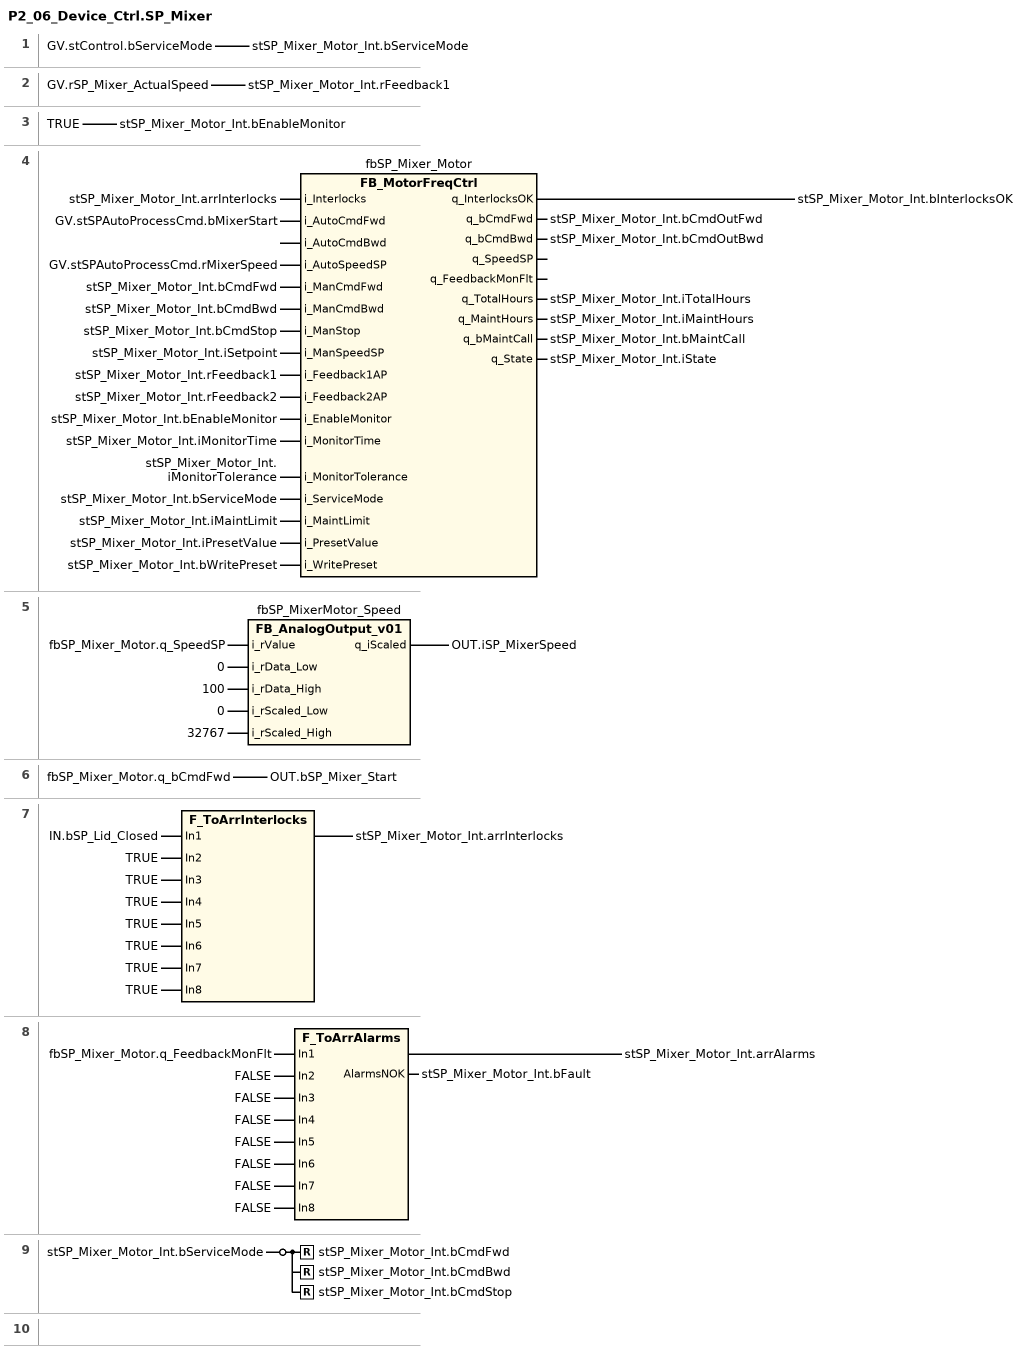
// NETWORK 1
stSP_Mixer_Motor_Int.bServiceMode := GV.stControl.bServiceMode;

// NETWORK 2
stSP_Mixer_Motor_Int.rFeedback1 := GV.rSP_Mixer_ActualSpeed;

// NETWORK 3
stSP_Mixer_Motor_Int.bEnableMonitor := TRUE;

// NETWORK 4
fbSP_Mixer_Motor(
    i_Interlocks := stSP_Mixer_Motor_Int.arrInterlocks,
    i_AutoCmdFwd := GV.stSPAutoProcessCmd.bMixerStart,
    i_AutoSpeedSP := GV.stSPAutoProcessCmd.rMixerSpeed,
    i_ManCmdFwd := stSP_Mixer_Motor_Int.bCmdFwd,
    i_ManCmdBwd := stSP_Mixer_Motor_Int.bCmdBwd,
    i_ManStop := stSP_Mixer_Motor_Int.bCmdStop,
    i_ManSpeedSP := stSP_Mixer_Motor_Int.iSetpoint,
    i_Feedback1AP := stSP_Mixer_Motor_Int.rFeedback1,
    i_Feedback2AP := stSP_Mixer_Motor_Int.rFeedback2,
    i_EnableMonitor := stSP_Mixer_Motor_Int.bEnableMonitor,
    i_MonitorTime := stSP_Mixer_Motor_Int.iMonitorTime,
    i_MonitorTolerance := stSP_Mixer_Motor_Int.iMonitorTolerance,
    i_ServiceMode := stSP_Mixer_Motor_Int.bServiceMode,
    i_MaintLimit := stSP_Mixer_Motor_Int.iMaintLimit,
    i_PresetValue := stSP_Mixer_Motor_Int.iPresetValue,
    i_WritePreset := stSP_Mixer_Motor_Int.bWritePreset,
    q_bCmdFwd => stSP_Mixer_Motor_Int.bCmdOutFwd,
    q_bCmdBwd => stSP_Mixer_Motor_Int.bCmdOutBwd,
    q_TotalHours => stSP_Mixer_Motor_Int.iTotalHours,
    q_MaintHours => stSP_Mixer_Motor_Int.iMaintHours,
    q_bMaintCall => stSP_Mixer_Motor_Int.bMaintCall,
    q_State => stSP_Mixer_Motor_Int.iState); // FB_MotorFreqCtrl
stSP_Mixer_Motor_Int.bInterlocksOK := fbSP_Mixer_Motor.q_InterlocksOK;

// NETWORK 5
fbSP_MixerMotor_Speed(
    i_rValue := fbSP_Mixer_Motor.q_SpeedSP,
    i_rData_Low := 0,
    i_rData_High := 100,
    i_rScaled_Low := 0,
    i_rScaled_High := 32767); // FB_AnalogOutput_v01
OUT.iSP_MixerSpeed := fbSP_MixerMotor_Speed.q_iScaled;

// NETWORK 6
OUT.bSP_Mixer_Start := fbSP_Mixer_Motor.q_bCmdFwd;

// NETWORK 7
stSP_Mixer_Motor_Int.arrInterlocks := F_ToArrInterlocks(In1 := IN.bSP_Lid_Closed, In2 := TRUE, In3 := TRUE, In4 := TRUE, In5 := TRUE, In6 := TRUE, In7 := TRUE, In8 := TRUE);

// NETWORK 8
stSP_Mixer_Motor_Int.arrAlarms := F_ToArrAlarms(In1 := fbSP_Mixer_Motor.q_FeedbackMonFlt, In2 := FALSE, In3 := FALSE, In4 := FALSE, In5 := FALSE, In6 := FALSE, In7 := FALSE, In8 := FALSE, AlarmsNOK => stSP_Mixer_Motor_Int.bFault);

// NETWORK 9
_w8 := NOT stSP_Mixer_Motor_Int.bServiceMode;
stSP_Mixer_Motor_Int.bCmdFwd R= _w8;
stSP_Mixer_Motor_Int.bCmdBwd R= _w8;
stSP_Mixer_Motor_Int.bCmdStop R= _w8;

// NETWORK 10
END_ACTION

ACTION SP_Pressure:
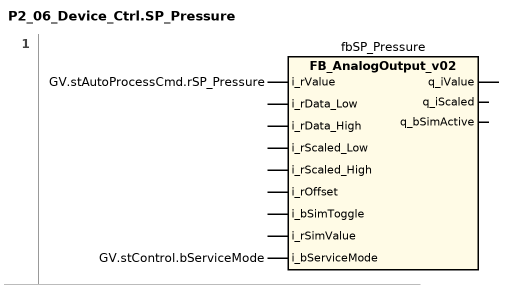
// NETWORK 1
fbSP_Pressure(i_rValue := GV.stAutoProcessCmd.rSP_Pressure, i_bServiceMode := GV.stControl.bServiceMode); // FB_AnalogOutput_v02
END_ACTION

ACTION SP_Temperature:
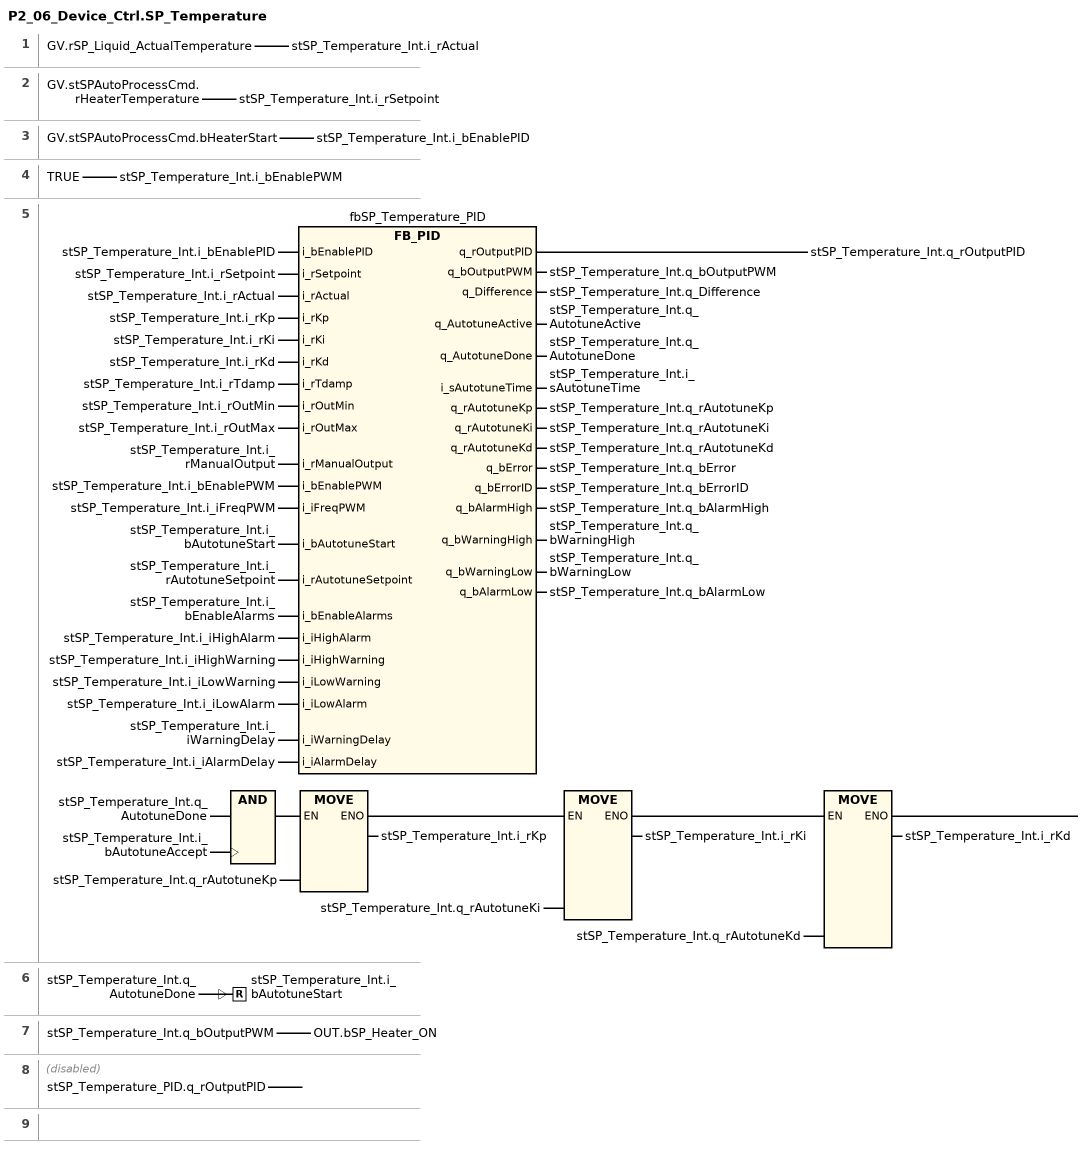
// NETWORK 1
stSP_Temperature_Int.i_rActual := GV.rSP_Liquid_ActualTemperature;

// NETWORK 2
stSP_Temperature_Int.i_rSetpoint := GV.stSPAutoProcessCmd.rHeaterTemperature;

// NETWORK 3
stSP_Temperature_Int.i_bEnablePID := GV.stSPAutoProcessCmd.bHeaterStart;

// NETWORK 4
stSP_Temperature_Int.i_bEnablePWM := TRUE;

// NETWORK 5
fbSP_Temperature_PID(
    i_bEnablePID := stSP_Temperature_Int.i_bEnablePID,
    i_rSetpoint := stSP_Temperature_Int.i_rSetpoint,
    i_rActual := stSP_Temperature_Int.i_rActual,
    i_rKp := stSP_Temperature_Int.i_rKp,
    i_rKi := stSP_Temperature_Int.i_rKi,
    i_rKd := stSP_Temperature_Int.i_rKd,
    i_rTdamp := stSP_Temperature_Int.i_rTdamp,
    i_rOutMin := stSP_Temperature_Int.i_rOutMin,
    i_rOutMax := stSP_Temperature_Int.i_rOutMax,
    i_rManualOutput := stSP_Temperature_Int.i_rManualOutput,
    i_bEnablePWM := stSP_Temperature_Int.i_bEnablePWM,
    i_iFreqPWM := stSP_Temperature_Int.i_iFreqPWM,
    i_bAutotuneStart := stSP_Temperature_Int.i_bAutotuneStart,
    i_rAutotuneSetpoint := stSP_Temperature_Int.i_rAutotuneSetpoint,
    i_bEnableAlarms := stSP_Temperature_Int.i_bEnableAlarms,
    i_iHighAlarm := stSP_Temperature_Int.i_iHighAlarm,
    i_iHighWarning := stSP_Temperature_Int.i_iHighWarning,
    i_iLowWarning := stSP_Temperature_Int.i_iLowWarning,
    i_iLowAlarm := stSP_Temperature_Int.i_iLowAlarm,
    i_iWarningDelay := stSP_Temperature_Int.i_iWarningDelay,
    i_iAlarmDelay := stSP_Temperature_Int.i_iAlarmDelay,
    q_bOutputPWM => stSP_Temperature_Int.q_bOutputPWM,
    q_Difference => stSP_Temperature_Int.q_Difference,
    q_AutotuneActive => stSP_Temperature_Int.q_AutotuneActive,
    q_AutotuneDone => stSP_Temperature_Int.q_AutotuneDone,
    i_sAutotuneTime => stSP_Temperature_Int.i_sAutotuneTime,
    q_rAutotuneKp => stSP_Temperature_Int.q_rAutotuneKp,
    q_rAutotuneKi => stSP_Temperature_Int.q_rAutotuneKi,
    q_rAutotuneKd => stSP_Temperature_Int.q_rAutotuneKd,
    q_bError => stSP_Temperature_Int.q_bError,
    q_bErrorID => stSP_Temperature_Int.q_bErrorID,
    q_bAlarmHigh => stSP_Temperature_Int.q_bAlarmHigh,
    q_bWarningHigh => stSP_Temperature_Int.q_bWarningHigh,
    q_bWarningLow => stSP_Temperature_Int.q_bWarningLow,
    q_bAlarmLow => stSP_Temperature_Int.q_bAlarmLow); // FB_PID
stSP_Temperature_Int.q_rOutputPID := fbSP_Temperature_PID.q_rOutputPID;
_rt1(CLK := stSP_Temperature_Int.i_bAutotuneAccept);
_w9 := stSP_Temperature_Int.q_AutotuneDone AND _rt1.Q;
IF _w9 THEN stSP_Temperature_Int.i_rKp := stSP_Temperature_Int.q_rAutotuneKp; END_IF
IF _w9 THEN stSP_Temperature_Int.i_rKi := stSP_Temperature_Int.q_rAutotuneKi; END_IF
IF _w9 THEN stSP_Temperature_Int.i_rKd := stSP_Temperature_Int.q_rAutotuneKd; END_IF

// NETWORK 6
_rt2(CLK := stSP_Temperature_Int.q_AutotuneDone);
stSP_Temperature_Int.i_bAutotuneStart R= _rt2.Q;

// NETWORK 7
OUT.bSP_Heater_ON := stSP_Temperature_Int.q_bOutputPWM;

// NETWORK 8 (disabled)
// ??? := stSP_Temperature_PID.q_rOutputPID;

// NETWORK 9
END_ACTION

ACTION Tool:
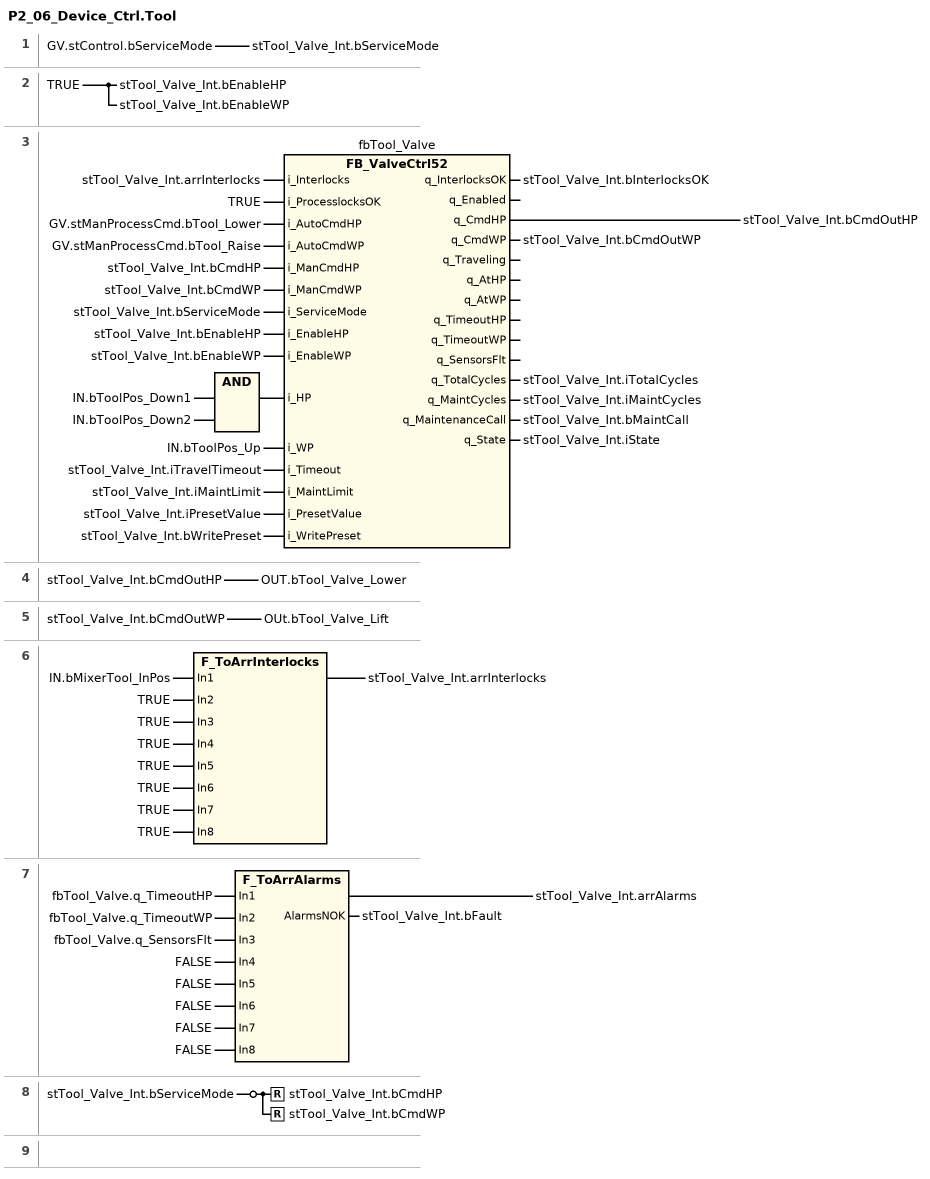
// NETWORK 1
stTool_Valve_Int.bServiceMode := GV.stControl.bServiceMode;

// NETWORK 2
stTool_Valve_Int.bEnableHP := TRUE;
stTool_Valve_Int.bEnableWP := TRUE;

// NETWORK 3
fbTool_Valve(
    i_Interlocks := stTool_Valve_Int.arrInterlocks,
    i_ProcesslocksOK := TRUE,
    i_AutoCmdHP := GV.stManProcessCmd.bTool_Lower,
    i_AutoCmdWP := GV.stManProcessCmd.bTool_Raise,
    i_ManCmdHP := stTool_Valve_Int.bCmdHP,
    i_ManCmdWP := stTool_Valve_Int.bCmdWP,
    i_ServiceMode := stTool_Valve_Int.bServiceMode,
    i_EnableHP := stTool_Valve_Int.bEnableHP,
    i_EnableWP := stTool_Valve_Int.bEnableWP,
    i_HP := IN.bToolPos_Down1 AND IN.bToolPos_Down2,
    i_WP := IN.bToolPos_Up,
    i_Timeout := stTool_Valve_Int.iTravelTimeout,
    i_MaintLimit := stTool_Valve_Int.iMaintLimit,
    i_PresetValue := stTool_Valve_Int.iPresetValue,
    i_WritePreset := stTool_Valve_Int.bWritePreset,
    q_InterlocksOK => stTool_Valve_Int.bInterlocksOK,
    q_CmdWP => stTool_Valve_Int.bCmdOutWP,
    q_TotalCycles => stTool_Valve_Int.iTotalCycles,
    q_MaintCycles => stTool_Valve_Int.iMaintCycles,
    q_MaintenanceCall => stTool_Valve_Int.bMaintCall,
    q_State => stTool_Valve_Int.iState); // FB_ValveCtrl52
stTool_Valve_Int.bCmdOutHP := fbTool_Valve.q_CmdHP;

// NETWORK 4
OUT.bTool_Valve_Lower := stTool_Valve_Int.bCmdOutHP;

// NETWORK 5
OUt.bTool_Valve_Lift := stTool_Valve_Int.bCmdOutWP;

// NETWORK 6
stTool_Valve_Int.arrInterlocks := F_ToArrInterlocks(In1 := IN.bMixerTool_InPos, In2 := TRUE, In3 := TRUE, In4 := TRUE, In5 := TRUE, In6 := TRUE, In7 := TRUE, In8 := TRUE);

// NETWORK 7
stTool_Valve_Int.arrAlarms := F_ToArrAlarms(In1 := fbTool_Valve.q_TimeoutHP, In2 := fbTool_Valve.q_TimeoutWP, In3 := fbTool_Valve.q_SensorsFlt, In4 := FALSE, In5 := FALSE, In6 := FALSE, In7 := FALSE, In8 := FALSE, AlarmsNOK => stTool_Valve_Int.bFault);

// NETWORK 8
_w10 := NOT stTool_Valve_Int.bServiceMode;
stTool_Valve_Int.bCmdHP R= _w10;
stTool_Valve_Int.bCmdWP R= _w10;

// NETWORK 9
END_ACTION

ACTION WIP_Chopper:
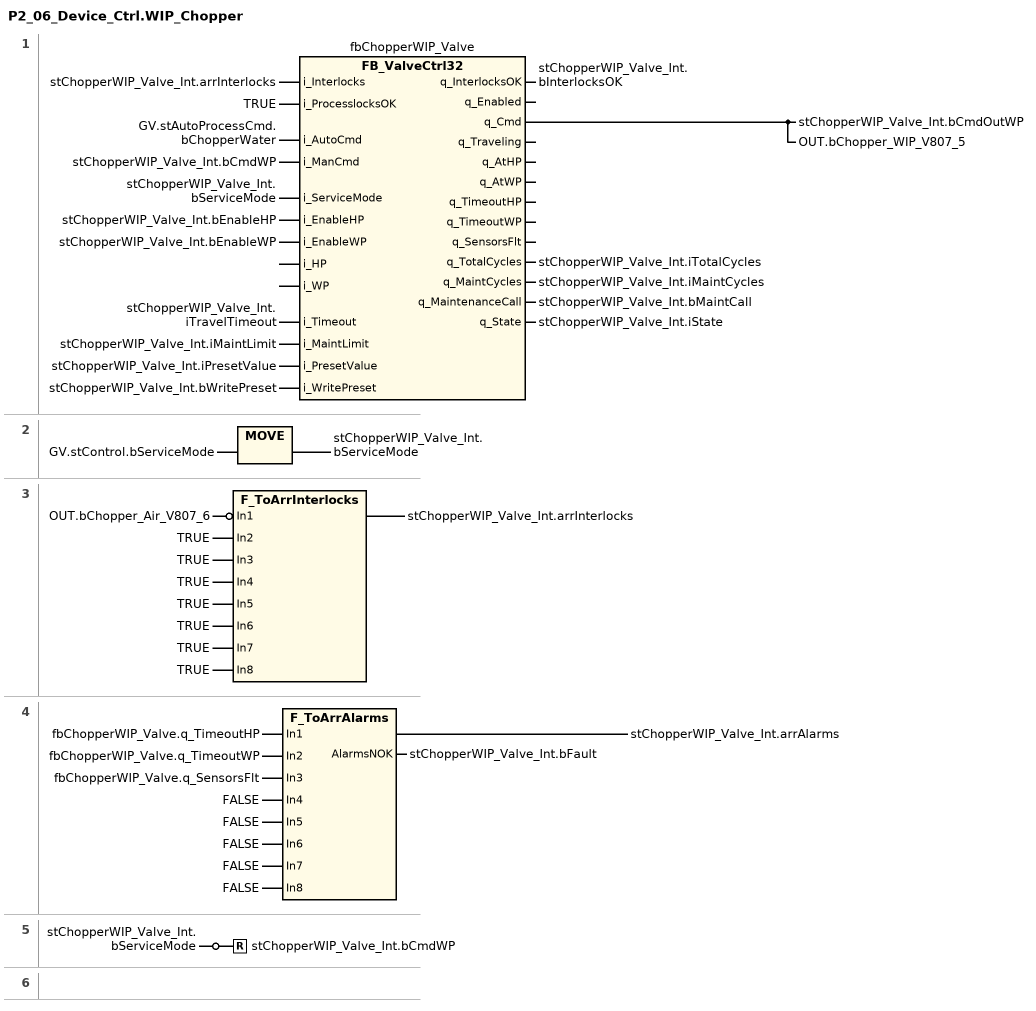
// NETWORK 1
fbChopperWIP_Valve(
    i_Interlocks := stChopperWIP_Valve_Int.arrInterlocks,
    i_ProcesslocksOK := TRUE,
    i_AutoCmd := GV.stAutoProcessCmd.bChopperWater,
    i_ManCmd := stChopperWIP_Valve_Int.bCmdWP,
    i_ServiceMode := stChopperWIP_Valve_Int.bServiceMode,
    i_EnableHP := stChopperWIP_Valve_Int.bEnableHP,
    i_EnableWP := stChopperWIP_Valve_Int.bEnableWP,
    i_Timeout := stChopperWIP_Valve_Int.iTravelTimeout,
    i_MaintLimit := stChopperWIP_Valve_Int.iMaintLimit,
    i_PresetValue := stChopperWIP_Valve_Int.iPresetValue,
    i_WritePreset := stChopperWIP_Valve_Int.bWritePreset,
    q_InterlocksOK => stChopperWIP_Valve_Int.bInterlocksOK,
    q_TotalCycles => stChopperWIP_Valve_Int.iTotalCycles,
    q_MaintCycles => stChopperWIP_Valve_Int.iMaintCycles,
    q_MaintenanceCall => stChopperWIP_Valve_Int.bMaintCall,
    q_State => stChopperWIP_Valve_Int.iState); // FB_ValveCtrl32
stChopperWIP_Valve_Int.bCmdOutWP := fbChopperWIP_Valve.q_Cmd;
OUT.bChopper_WIP_V807_5 := fbChopperWIP_Valve.q_Cmd;

// NETWORK 2
stChopperWIP_Valve_Int.bServiceMode := GV.stControl.bServiceMode;

// NETWORK 3
stChopperWIP_Valve_Int.arrInterlocks := F_ToArrInterlocks(In1 := NOT OUT.bChopper_Air_V807_6, In2 := TRUE, In3 := TRUE, In4 := TRUE, In5 := TRUE, In6 := TRUE, In7 := TRUE, In8 := TRUE);

// NETWORK 4
stChopperWIP_Valve_Int.arrAlarms := F_ToArrAlarms(In1 := fbChopperWIP_Valve.q_TimeoutHP, In2 := fbChopperWIP_Valve.q_TimeoutWP, In3 := fbChopperWIP_Valve.q_SensorsFlt, In4 := FALSE, In5 := FALSE, In6 := FALSE, In7 := FALSE, In8 := FALSE, AlarmsNOK => stChopperWIP_Valve_Int.bFault);

// NETWORK 5
stChopperWIP_Valve_Int.bCmdWP R= NOT stChopperWIP_Valve_Int.bServiceMode;

// NETWORK 6
END_ACTION

ACTION WIP_CleaningAir:
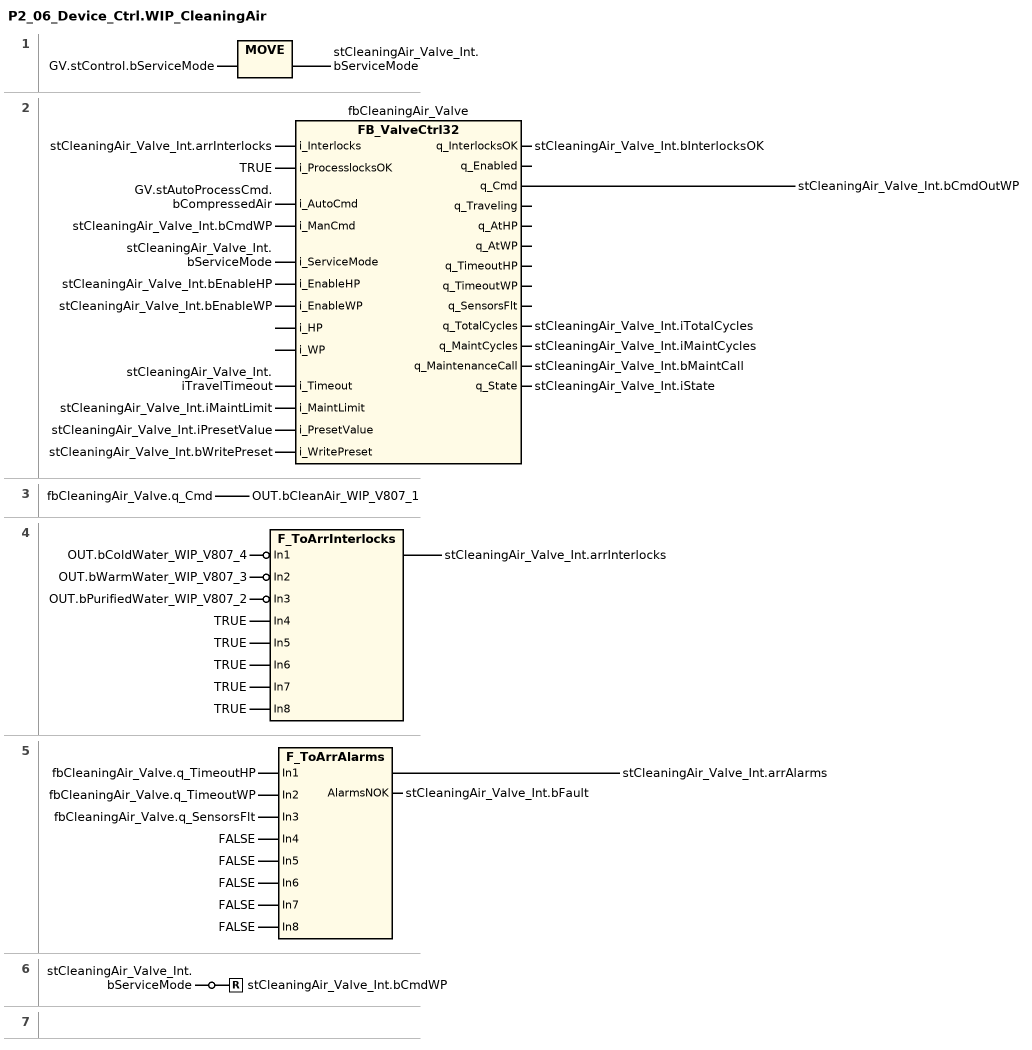
// NETWORK 1
stCleaningAir_Valve_Int.bServiceMode := GV.stControl.bServiceMode;

// NETWORK 2
fbCleaningAir_Valve(
    i_Interlocks := stCleaningAir_Valve_Int.arrInterlocks,
    i_ProcesslocksOK := TRUE,
    i_AutoCmd := GV.stAutoProcessCmd.bCompressedAir,
    i_ManCmd := stCleaningAir_Valve_Int.bCmdWP,
    i_ServiceMode := stCleaningAir_Valve_Int.bServiceMode,
    i_EnableHP := stCleaningAir_Valve_Int.bEnableHP,
    i_EnableWP := stCleaningAir_Valve_Int.bEnableWP,
    i_Timeout := stCleaningAir_Valve_Int.iTravelTimeout,
    i_MaintLimit := stCleaningAir_Valve_Int.iMaintLimit,
    i_PresetValue := stCleaningAir_Valve_Int.iPresetValue,
    i_WritePreset := stCleaningAir_Valve_Int.bWritePreset,
    q_InterlocksOK => stCleaningAir_Valve_Int.bInterlocksOK,
    q_TotalCycles => stCleaningAir_Valve_Int.iTotalCycles,
    q_MaintCycles => stCleaningAir_Valve_Int.iMaintCycles,
    q_MaintenanceCall => stCleaningAir_Valve_Int.bMaintCall,
    q_State => stCleaningAir_Valve_Int.iState); // FB_ValveCtrl32
stCleaningAir_Valve_Int.bCmdOutWP := fbCleaningAir_Valve.q_Cmd;

// NETWORK 3
OUT.bCleanAir_WIP_V807_1 := fbCleaningAir_Valve.q_Cmd;

// NETWORK 4
stCleaningAir_Valve_Int.arrInterlocks := F_ToArrInterlocks(In1 := NOT OUT.bColdWater_WIP_V807_4, In2 := NOT OUT.bWarmWater_WIP_V807_3, In3 := NOT OUT.bPurifiedWater_WIP_V807_2, In4 := TRUE, In5 := TRUE, In6 := TRUE, In7 := TRUE, In8 := TRUE);

// NETWORK 5
stCleaningAir_Valve_Int.arrAlarms := F_ToArrAlarms(In1 := fbCleaningAir_Valve.q_TimeoutHP, In2 := fbCleaningAir_Valve.q_TimeoutWP, In3 := fbCleaningAir_Valve.q_SensorsFlt, In4 := FALSE, In5 := FALSE, In6 := FALSE, In7 := FALSE, In8 := FALSE, AlarmsNOK => stCleaningAir_Valve_Int.bFault);

// NETWORK 6
stCleaningAir_Valve_Int.bCmdWP R= NOT stCleaningAir_Valve_Int.bServiceMode;

// NETWORK 7
END_ACTION

ACTION WIP_ColdWater:
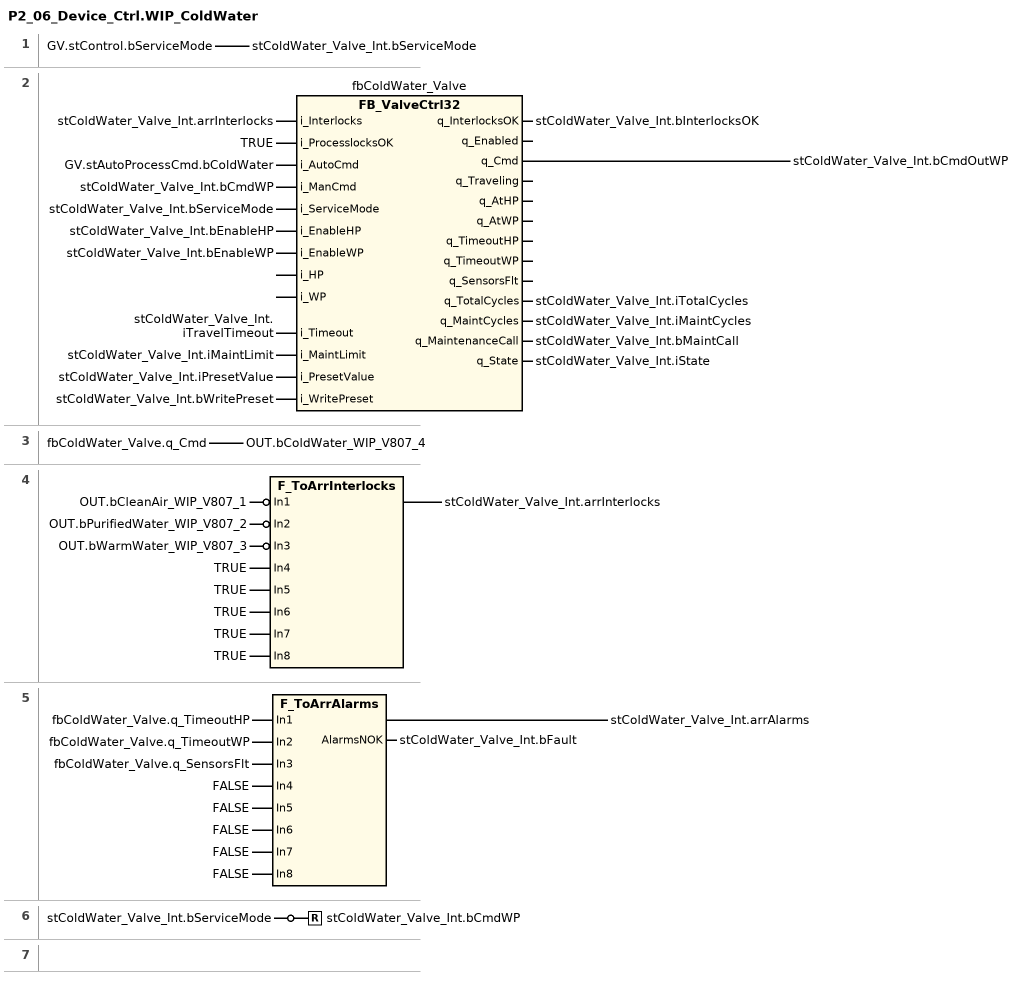
// NETWORK 1
stColdWater_Valve_Int.bServiceMode := GV.stControl.bServiceMode;

// NETWORK 2
fbColdWater_Valve(
    i_Interlocks := stColdWater_Valve_Int.arrInterlocks,
    i_ProcesslocksOK := TRUE,
    i_AutoCmd := GV.stAutoProcessCmd.bColdWater,
    i_ManCmd := stColdWater_Valve_Int.bCmdWP,
    i_ServiceMode := stColdWater_Valve_Int.bServiceMode,
    i_EnableHP := stColdWater_Valve_Int.bEnableHP,
    i_EnableWP := stColdWater_Valve_Int.bEnableWP,
    i_Timeout := stColdWater_Valve_Int.iTravelTimeout,
    i_MaintLimit := stColdWater_Valve_Int.iMaintLimit,
    i_PresetValue := stColdWater_Valve_Int.iPresetValue,
    i_WritePreset := stColdWater_Valve_Int.bWritePreset,
    q_InterlocksOK => stColdWater_Valve_Int.bInterlocksOK,
    q_TotalCycles => stColdWater_Valve_Int.iTotalCycles,
    q_MaintCycles => stColdWater_Valve_Int.iMaintCycles,
    q_MaintenanceCall => stColdWater_Valve_Int.bMaintCall,
    q_State => stColdWater_Valve_Int.iState); // FB_ValveCtrl32
stColdWater_Valve_Int.bCmdOutWP := fbColdWater_Valve.q_Cmd;

// NETWORK 3
OUT.bColdWater_WIP_V807_4 := fbColdWater_Valve.q_Cmd;

// NETWORK 4
stColdWater_Valve_Int.arrInterlocks := F_ToArrInterlocks(In1 := NOT OUT.bCleanAir_WIP_V807_1, In2 := NOT OUT.bPurifiedWater_WIP_V807_2, In3 := NOT OUT.bWarmWater_WIP_V807_3, In4 := TRUE, In5 := TRUE, In6 := TRUE, In7 := TRUE, In8 := TRUE);

// NETWORK 5
stColdWater_Valve_Int.arrAlarms := F_ToArrAlarms(In1 := fbColdWater_Valve.q_TimeoutHP, In2 := fbColdWater_Valve.q_TimeoutWP, In3 := fbColdWater_Valve.q_SensorsFlt, In4 := FALSE, In5 := FALSE, In6 := FALSE, In7 := FALSE, In8 := FALSE, AlarmsNOK => stColdWater_Valve_Int.bFault);

// NETWORK 6
stColdWater_Valve_Int.bCmdWP R= NOT stColdWater_Valve_Int.bServiceMode;

// NETWORK 7
END_ACTION

ACTION WIP_MainDrain:
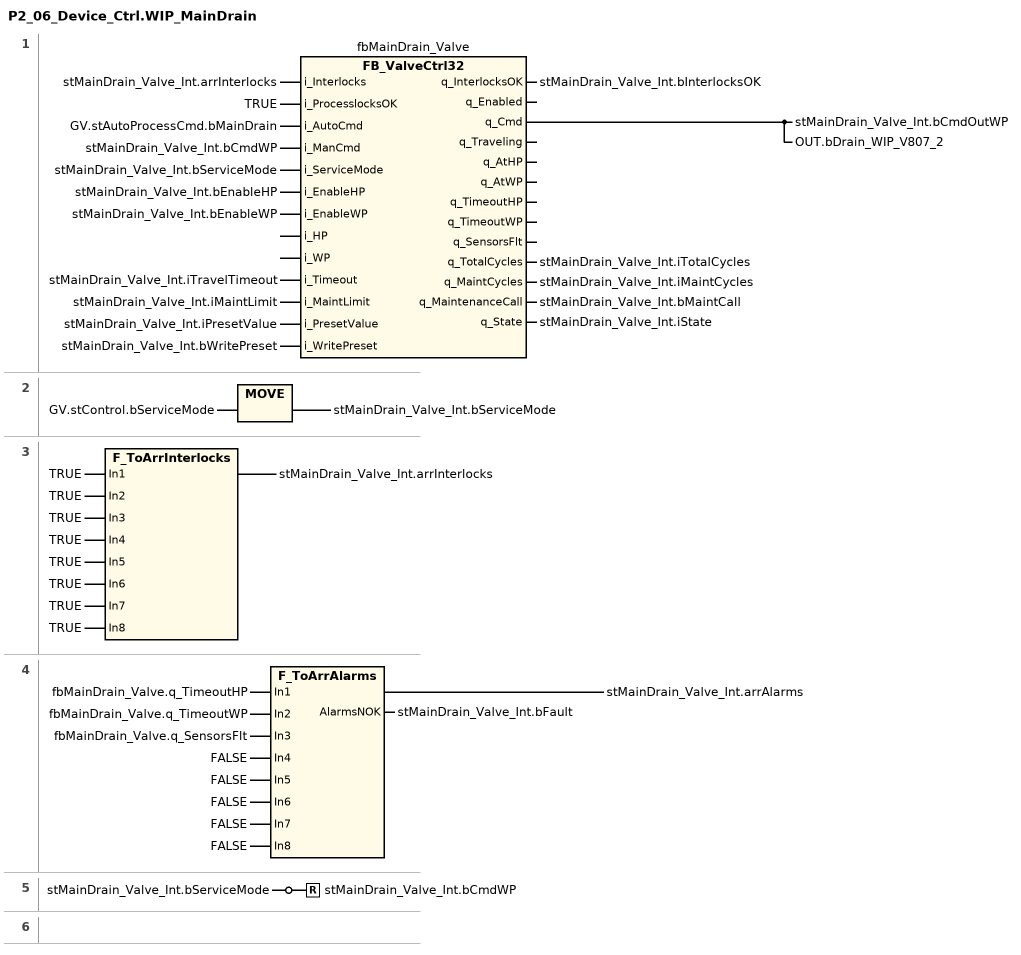
// NETWORK 1
fbMainDrain_Valve(
    i_Interlocks := stMainDrain_Valve_Int.arrInterlocks,
    i_ProcesslocksOK := TRUE,
    i_AutoCmd := GV.stAutoProcessCmd.bMainDrain,
    i_ManCmd := stMainDrain_Valve_Int.bCmdWP,
    i_ServiceMode := stMainDrain_Valve_Int.bServiceMode,
    i_EnableHP := stMainDrain_Valve_Int.bEnableHP,
    i_EnableWP := stMainDrain_Valve_Int.bEnableWP,
    i_Timeout := stMainDrain_Valve_Int.iTravelTimeout,
    i_MaintLimit := stMainDrain_Valve_Int.iMaintLimit,
    i_PresetValue := stMainDrain_Valve_Int.iPresetValue,
    i_WritePreset := stMainDrain_Valve_Int.bWritePreset,
    q_InterlocksOK => stMainDrain_Valve_Int.bInterlocksOK,
    q_TotalCycles => stMainDrain_Valve_Int.iTotalCycles,
    q_MaintCycles => stMainDrain_Valve_Int.iMaintCycles,
    q_MaintenanceCall => stMainDrain_Valve_Int.bMaintCall,
    q_State => stMainDrain_Valve_Int.iState); // FB_ValveCtrl32
stMainDrain_Valve_Int.bCmdOutWP := fbMainDrain_Valve.q_Cmd;
OUT.bDrain_WIP_V807_2 := fbMainDrain_Valve.q_Cmd;

// NETWORK 2
stMainDrain_Valve_Int.bServiceMode := GV.stControl.bServiceMode;

// NETWORK 3
stMainDrain_Valve_Int.arrInterlocks := F_ToArrInterlocks(In1 := TRUE, In2 := TRUE, In3 := TRUE, In4 := TRUE, In5 := TRUE, In6 := TRUE, In7 := TRUE, In8 := TRUE);

// NETWORK 4
stMainDrain_Valve_Int.arrAlarms := F_ToArrAlarms(In1 := fbMainDrain_Valve.q_TimeoutHP, In2 := fbMainDrain_Valve.q_TimeoutWP, In3 := fbMainDrain_Valve.q_SensorsFlt, In4 := FALSE, In5 := FALSE, In6 := FALSE, In7 := FALSE, In8 := FALSE, AlarmsNOK => stMainDrain_Valve_Int.bFault);

// NETWORK 5
stMainDrain_Valve_Int.bCmdWP R= NOT stMainDrain_Valve_Int.bServiceMode;

// NETWORK 6
END_ACTION

ACTION WIP_Mixer:
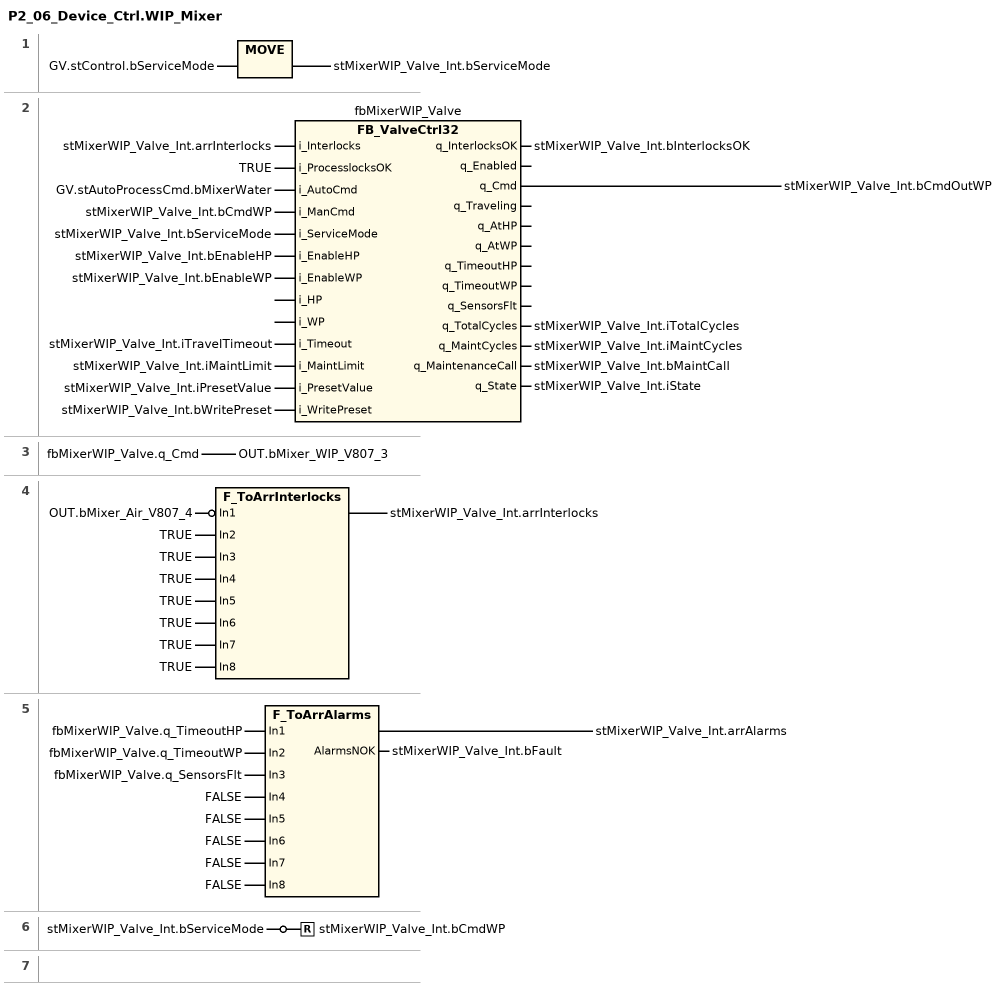
// NETWORK 1
stMixerWIP_Valve_Int.bServiceMode := GV.stControl.bServiceMode;

// NETWORK 2
fbMixerWIP_Valve(
    i_Interlocks := stMixerWIP_Valve_Int.arrInterlocks,
    i_ProcesslocksOK := TRUE,
    i_AutoCmd := GV.stAutoProcessCmd.bMixerWater,
    i_ManCmd := stMixerWIP_Valve_Int.bCmdWP,
    i_ServiceMode := stMixerWIP_Valve_Int.bServiceMode,
    i_EnableHP := stMixerWIP_Valve_Int.bEnableHP,
    i_EnableWP := stMixerWIP_Valve_Int.bEnableWP,
    i_Timeout := stMixerWIP_Valve_Int.iTravelTimeout,
    i_MaintLimit := stMixerWIP_Valve_Int.iMaintLimit,
    i_PresetValue := stMixerWIP_Valve_Int.iPresetValue,
    i_WritePreset := stMixerWIP_Valve_Int.bWritePreset,
    q_InterlocksOK => stMixerWIP_Valve_Int.bInterlocksOK,
    q_TotalCycles => stMixerWIP_Valve_Int.iTotalCycles,
    q_MaintCycles => stMixerWIP_Valve_Int.iMaintCycles,
    q_MaintenanceCall => stMixerWIP_Valve_Int.bMaintCall,
    q_State => stMixerWIP_Valve_Int.iState); // FB_ValveCtrl32
stMixerWIP_Valve_Int.bCmdOutWP := fbMixerWIP_Valve.q_Cmd;

// NETWORK 3
OUT.bMixer_WIP_V807_3 := fbMixerWIP_Valve.q_Cmd;

// NETWORK 4
stMixerWIP_Valve_Int.arrInterlocks := F_ToArrInterlocks(In1 := NOT OUT.bMixer_Air_V807_4, In2 := TRUE, In3 := TRUE, In4 := TRUE, In5 := TRUE, In6 := TRUE, In7 := TRUE, In8 := TRUE);

// NETWORK 5
stMixerWIP_Valve_Int.arrAlarms := F_ToArrAlarms(In1 := fbMixerWIP_Valve.q_TimeoutHP, In2 := fbMixerWIP_Valve.q_TimeoutWP, In3 := fbMixerWIP_Valve.q_SensorsFlt, In4 := FALSE, In5 := FALSE, In6 := FALSE, In7 := FALSE, In8 := FALSE, AlarmsNOK => stMixerWIP_Valve_Int.bFault);

// NETWORK 6
stMixerWIP_Valve_Int.bCmdWP R= NOT stMixerWIP_Valve_Int.bServiceMode;

// NETWORK 7
END_ACTION

ACTION WIP_PurifiedWater:
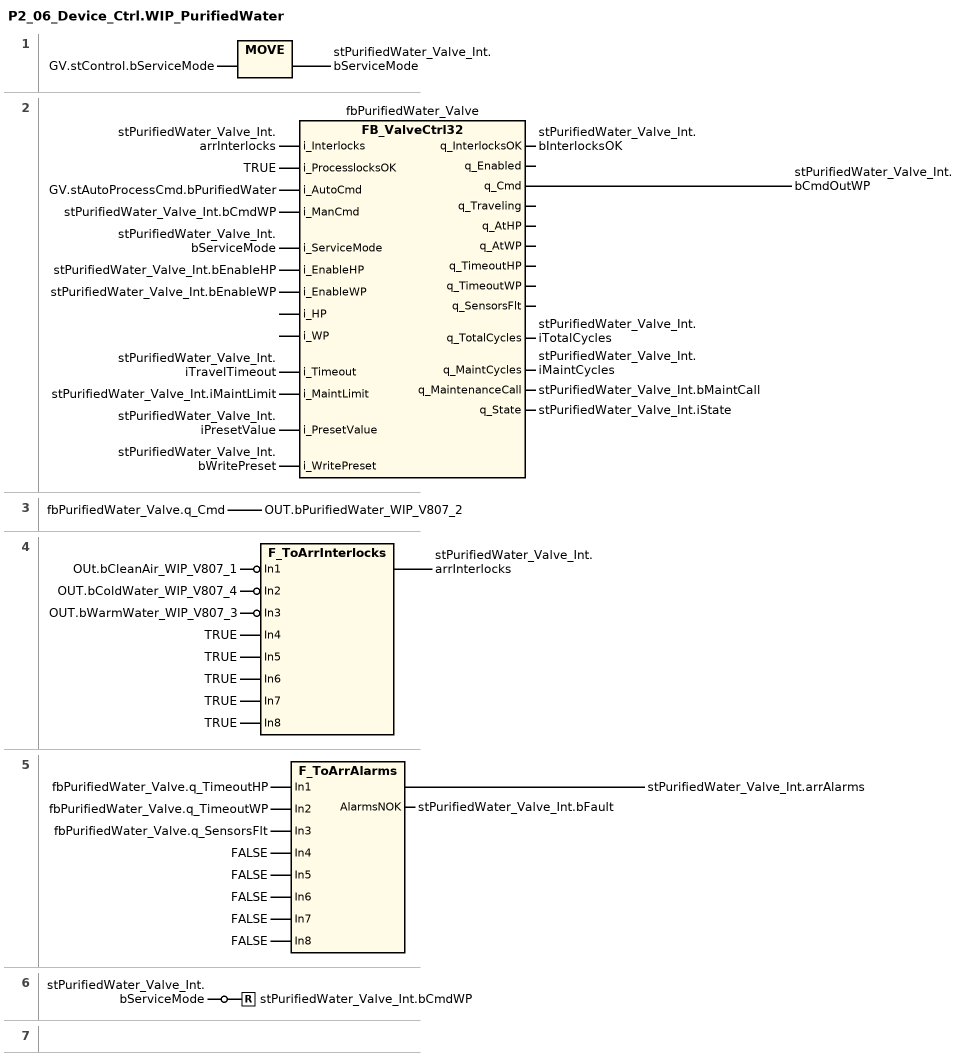
// NETWORK 1
stPurifiedWater_Valve_Int.bServiceMode := GV.stControl.bServiceMode;

// NETWORK 2
fbPurifiedWater_Valve(
    i_Interlocks := stPurifiedWater_Valve_Int.arrInterlocks,
    i_ProcesslocksOK := TRUE,
    i_AutoCmd := GV.stAutoProcessCmd.bPurifiedWater,
    i_ManCmd := stPurifiedWater_Valve_Int.bCmdWP,
    i_ServiceMode := stPurifiedWater_Valve_Int.bServiceMode,
    i_EnableHP := stPurifiedWater_Valve_Int.bEnableHP,
    i_EnableWP := stPurifiedWater_Valve_Int.bEnableWP,
    i_Timeout := stPurifiedWater_Valve_Int.iTravelTimeout,
    i_MaintLimit := stPurifiedWater_Valve_Int.iMaintLimit,
    i_PresetValue := stPurifiedWater_Valve_Int.iPresetValue,
    i_WritePreset := stPurifiedWater_Valve_Int.bWritePreset,
    q_InterlocksOK => stPurifiedWater_Valve_Int.bInterlocksOK,
    q_TotalCycles => stPurifiedWater_Valve_Int.iTotalCycles,
    q_MaintCycles => stPurifiedWater_Valve_Int.iMaintCycles,
    q_MaintenanceCall => stPurifiedWater_Valve_Int.bMaintCall,
    q_State => stPurifiedWater_Valve_Int.iState); // FB_ValveCtrl32
stPurifiedWater_Valve_Int.bCmdOutWP := fbPurifiedWater_Valve.q_Cmd;

// NETWORK 3
OUT.bPurifiedWater_WIP_V807_2 := fbPurifiedWater_Valve.q_Cmd;

// NETWORK 4
stPurifiedWater_Valve_Int.arrInterlocks := F_ToArrInterlocks(In1 := NOT OUt.bCleanAir_WIP_V807_1, In2 := NOT OUT.bColdWater_WIP_V807_4, In3 := NOT OUT.bWarmWater_WIP_V807_3, In4 := TRUE, In5 := TRUE, In6 := TRUE, In7 := TRUE, In8 := TRUE);

// NETWORK 5
stPurifiedWater_Valve_Int.arrAlarms := F_ToArrAlarms(In1 := fbPurifiedWater_Valve.q_TimeoutHP, In2 := fbPurifiedWater_Valve.q_TimeoutWP, In3 := fbPurifiedWater_Valve.q_SensorsFlt, In4 := FALSE, In5 := FALSE, In6 := FALSE, In7 := FALSE, In8 := FALSE, AlarmsNOK => stPurifiedWater_Valve_Int.bFault);

// NETWORK 6
stPurifiedWater_Valve_Int.bCmdWP R= NOT stPurifiedWater_Valve_Int.bServiceMode;

// NETWORK 7
END_ACTION

ACTION WIP_SP:
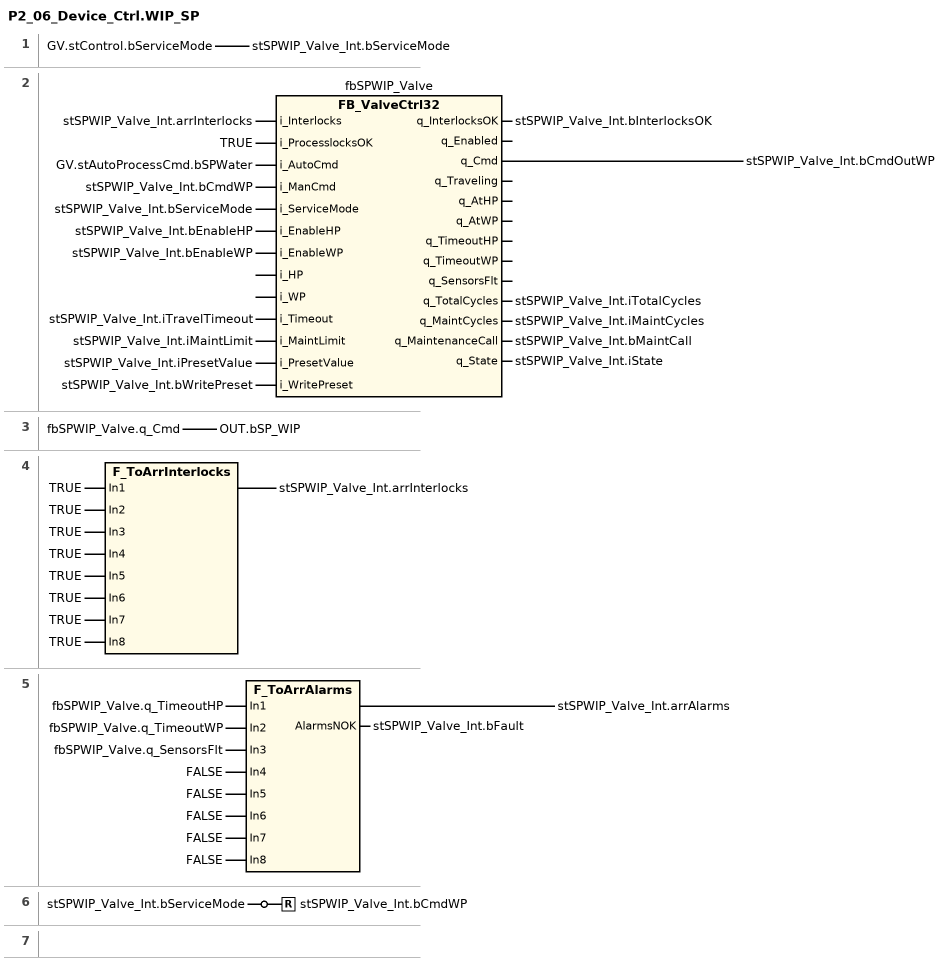
// NETWORK 1
stSPWIP_Valve_Int.bServiceMode := GV.stControl.bServiceMode;

// NETWORK 2
fbSPWIP_Valve(
    i_Interlocks := stSPWIP_Valve_Int.arrInterlocks,
    i_ProcesslocksOK := TRUE,
    i_AutoCmd := GV.stAutoProcessCmd.bSPWater,
    i_ManCmd := stSPWIP_Valve_Int.bCmdWP,
    i_ServiceMode := stSPWIP_Valve_Int.bServiceMode,
    i_EnableHP := stSPWIP_Valve_Int.bEnableHP,
    i_EnableWP := stSPWIP_Valve_Int.bEnableWP,
    i_Timeout := stSPWIP_Valve_Int.iTravelTimeout,
    i_MaintLimit := stSPWIP_Valve_Int.iMaintLimit,
    i_PresetValue := stSPWIP_Valve_Int.iPresetValue,
    i_WritePreset := stSPWIP_Valve_Int.bWritePreset,
    q_InterlocksOK => stSPWIP_Valve_Int.bInterlocksOK,
    q_TotalCycles => stSPWIP_Valve_Int.iTotalCycles,
    q_MaintCycles => stSPWIP_Valve_Int.iMaintCycles,
    q_MaintenanceCall => stSPWIP_Valve_Int.bMaintCall,
    q_State => stSPWIP_Valve_Int.iState); // FB_ValveCtrl32
stSPWIP_Valve_Int.bCmdOutWP := fbSPWIP_Valve.q_Cmd;

// NETWORK 3
OUT.bSP_WIP := fbSPWIP_Valve.q_Cmd;

// NETWORK 4
stSPWIP_Valve_Int.arrInterlocks := F_ToArrInterlocks(In1 := TRUE, In2 := TRUE, In3 := TRUE, In4 := TRUE, In5 := TRUE, In6 := TRUE, In7 := TRUE, In8 := TRUE);

// NETWORK 5
stSPWIP_Valve_Int.arrAlarms := F_ToArrAlarms(In1 := fbSPWIP_Valve.q_TimeoutHP, In2 := fbSPWIP_Valve.q_TimeoutWP, In3 := fbSPWIP_Valve.q_SensorsFlt, In4 := FALSE, In5 := FALSE, In6 := FALSE, In7 := FALSE, In8 := FALSE, AlarmsNOK => stSPWIP_Valve_Int.bFault);

// NETWORK 6
stSPWIP_Valve_Int.bCmdWP R= NOT stSPWIP_Valve_Int.bServiceMode;

// NETWORK 7
END_ACTION

ACTION WIP_SPDrain:
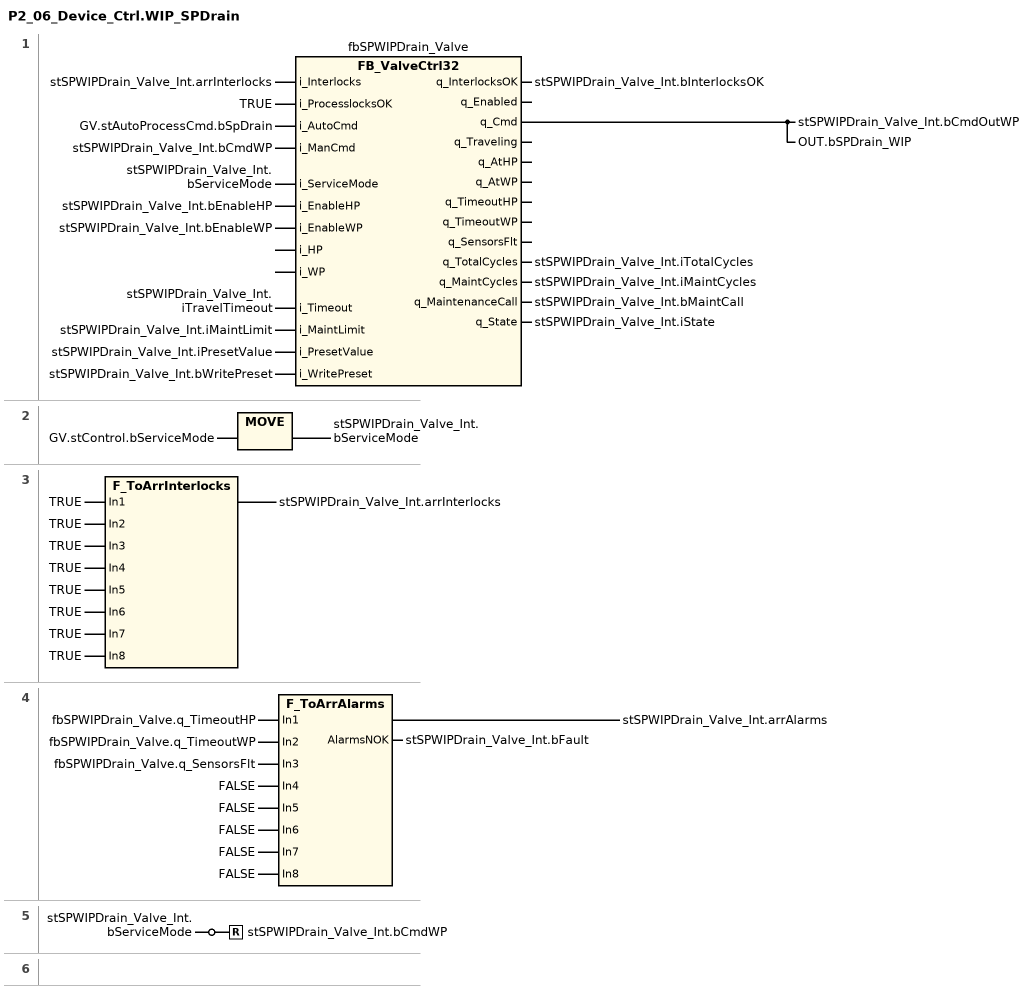
// NETWORK 1
fbSPWIPDrain_Valve(
    i_Interlocks := stSPWIPDrain_Valve_Int.arrInterlocks,
    i_ProcesslocksOK := TRUE,
    i_AutoCmd := GV.stAutoProcessCmd.bSpDrain,
    i_ManCmd := stSPWIPDrain_Valve_Int.bCmdWP,
    i_ServiceMode := stSPWIPDrain_Valve_Int.bServiceMode,
    i_EnableHP := stSPWIPDrain_Valve_Int.bEnableHP,
    i_EnableWP := stSPWIPDrain_Valve_Int.bEnableWP,
    i_Timeout := stSPWIPDrain_Valve_Int.iTravelTimeout,
    i_MaintLimit := stSPWIPDrain_Valve_Int.iMaintLimit,
    i_PresetValue := stSPWIPDrain_Valve_Int.iPresetValue,
    i_WritePreset := stSPWIPDrain_Valve_Int.bWritePreset,
    q_InterlocksOK => stSPWIPDrain_Valve_Int.bInterlocksOK,
    q_TotalCycles => stSPWIPDrain_Valve_Int.iTotalCycles,
    q_MaintCycles => stSPWIPDrain_Valve_Int.iMaintCycles,
    q_MaintenanceCall => stSPWIPDrain_Valve_Int.bMaintCall,
    q_State => stSPWIPDrain_Valve_Int.iState); // FB_ValveCtrl32
stSPWIPDrain_Valve_Int.bCmdOutWP := fbSPWIPDrain_Valve.q_Cmd;
OUT.bSPDrain_WIP := fbSPWIPDrain_Valve.q_Cmd;

// NETWORK 2
stSPWIPDrain_Valve_Int.bServiceMode := GV.stControl.bServiceMode;

// NETWORK 3
stSPWIPDrain_Valve_Int.arrInterlocks := F_ToArrInterlocks(In1 := TRUE, In2 := TRUE, In3 := TRUE, In4 := TRUE, In5 := TRUE, In6 := TRUE, In7 := TRUE, In8 := TRUE);

// NETWORK 4
stSPWIPDrain_Valve_Int.arrAlarms := F_ToArrAlarms(In1 := fbSPWIPDrain_Valve.q_TimeoutHP, In2 := fbSPWIPDrain_Valve.q_TimeoutWP, In3 := fbSPWIPDrain_Valve.q_SensorsFlt, In4 := FALSE, In5 := FALSE, In6 := FALSE, In7 := FALSE, In8 := FALSE, AlarmsNOK => stSPWIPDrain_Valve_Int.bFault);

// NETWORK 5
stSPWIPDrain_Valve_Int.bCmdWP R= NOT stSPWIPDrain_Valve_Int.bServiceMode;

// NETWORK 6
END_ACTION

ACTION WIP_WarmWater:
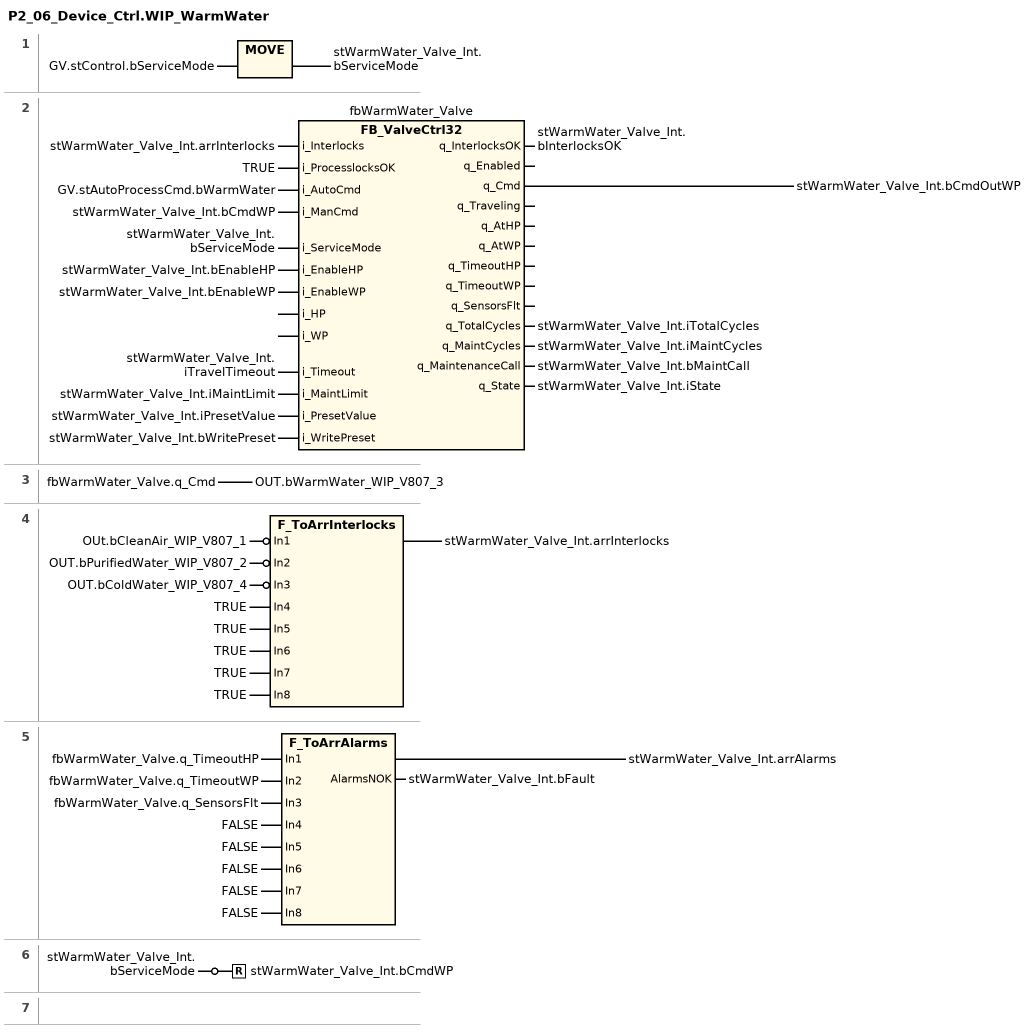
// NETWORK 1
stWarmWater_Valve_Int.bServiceMode := GV.stControl.bServiceMode;

// NETWORK 2
fbWarmWater_Valve(
    i_Interlocks := stWarmWater_Valve_Int.arrInterlocks,
    i_ProcesslocksOK := TRUE,
    i_AutoCmd := GV.stAutoProcessCmd.bWarmWater,
    i_ManCmd := stWarmWater_Valve_Int.bCmdWP,
    i_ServiceMode := stWarmWater_Valve_Int.bServiceMode,
    i_EnableHP := stWarmWater_Valve_Int.bEnableHP,
    i_EnableWP := stWarmWater_Valve_Int.bEnableWP,
    i_Timeout := stWarmWater_Valve_Int.iTravelTimeout,
    i_MaintLimit := stWarmWater_Valve_Int.iMaintLimit,
    i_PresetValue := stWarmWater_Valve_Int.iPresetValue,
    i_WritePreset := stWarmWater_Valve_Int.bWritePreset,
    q_InterlocksOK => stWarmWater_Valve_Int.bInterlocksOK,
    q_TotalCycles => stWarmWater_Valve_Int.iTotalCycles,
    q_MaintCycles => stWarmWater_Valve_Int.iMaintCycles,
    q_MaintenanceCall => stWarmWater_Valve_Int.bMaintCall,
    q_State => stWarmWater_Valve_Int.iState); // FB_ValveCtrl32
stWarmWater_Valve_Int.bCmdOutWP := fbWarmWater_Valve.q_Cmd;

// NETWORK 3
OUT.bWarmWater_WIP_V807_3 := fbWarmWater_Valve.q_Cmd;

// NETWORK 4
stWarmWater_Valve_Int.arrInterlocks := F_ToArrInterlocks(In1 := NOT OUt.bCleanAir_WIP_V807_1, In2 := NOT OUT.bPurifiedWater_WIP_V807_2, In3 := NOT OUT.bColdWater_WIP_V807_4, In4 := TRUE, In5 := TRUE, In6 := TRUE, In7 := TRUE, In8 := TRUE);

// NETWORK 5
stWarmWater_Valve_Int.arrAlarms := F_ToArrAlarms(In1 := fbWarmWater_Valve.q_TimeoutHP, In2 := fbWarmWater_Valve.q_TimeoutWP, In3 := fbWarmWater_Valve.q_SensorsFlt, In4 := FALSE, In5 := FALSE, In6 := FALSE, In7 := FALSE, In8 := FALSE, AlarmsNOK => stWarmWater_Valve_Int.bFault);

// NETWORK 6
stWarmWater_Valve_Int.bCmdWP R= NOT stWarmWater_Valve_Int.bServiceMode;

// NETWORK 7
END_ACTION

END_PROGRAM

// ---- FBs/Devices/FB_MotorFreqCtrl.TcPOU
FUNCTION_BLOCK FB_MotorFreqCtrl
VAR_INPUT
	i_Interlocks		:ARRAY[1..8] OF BOOL;
	i_AutoCmdFwd		:BOOL;
	i_AutoCmdBwd		:BOOL;
	i_AutoSpeedSP		:REAL;
	i_ManCmdFwd			:BOOL;
	i_ManCmdBwd			:BOOL;
	i_ManStop			:BOOL;
	i_ManSpeedSP		:REAL;
	i_Feedback1AP		:REAL;
	i_Feedback2AP		:REAL;
	i_EnableMonitor		:BOOL;
	i_MonitorTime		:INT;
	i_MonitorTolerance	:INT;
	i_ServiceMode		:BOOL;
	i_MaintLimit		:REAL;
	i_PresetValue		:REAL;
	i_WritePreset		:BOOL;
END_VAR
VAR_OUTPUT
	q_InterlocksOK		:BOOL;
	q_bCmdFwd			:BOOL;
	q_bCmdBwd			:BOOL;
	q_SpeedSP			:REAL;
	q_FeedbackMonFlt	:BOOL;
	q_TotalHours		:REAL;
	q_MaintHours		:REAL;
	q_bMaintCall		:BOOL;	
	q_State				:INT;
END_VAR
VAR
	bCmdFwd				:BOOL;
	bCmdBwd				:BOOL;
	tRunTime			:TIME;
	tRunTime1			:TIME;
	rRunTime			:REAL;
	tofCMDFwd			:TOF;
	tofCMDBwd			:TOF;
	tonFwdOff			:TON;
	tonBcwOff			:TON;
	tonMonFdb			:TON;
	tonMotorRun			:TON;
	tofMotorRun			:TOF;
END_VAR
VAR // added by the converter: edge detectors and wires of the graphical bodies
    _w1, _w2 : BOOL;
    _ft1, _ft2 : F_TRIG;
    _rt1 : R_TRIG;
END_VAR

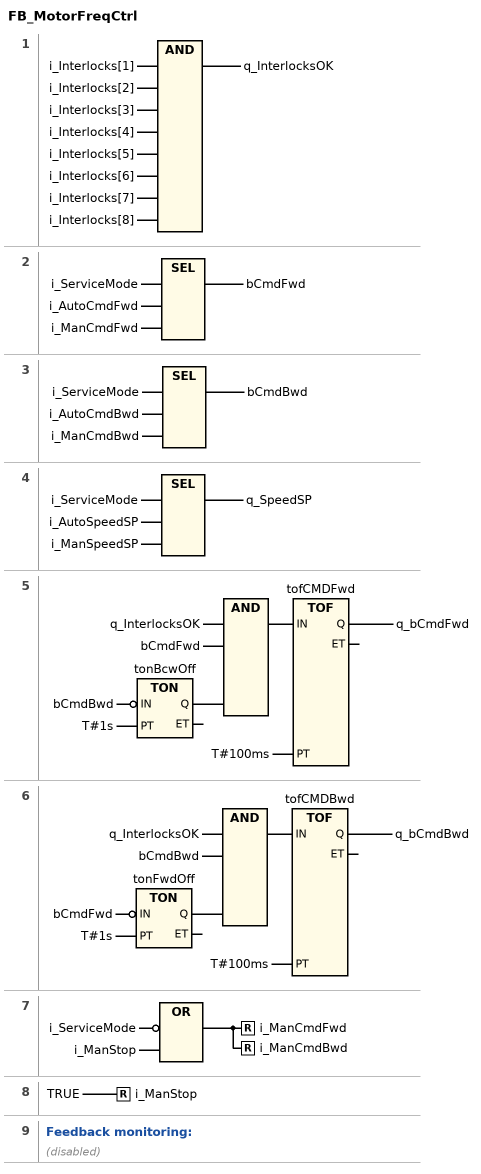
// NETWORK 1
q_InterlocksOK := i_Interlocks[1] AND i_Interlocks[2] AND i_Interlocks[3] AND i_Interlocks[4] AND i_Interlocks[5] AND i_Interlocks[6] AND i_Interlocks[7] AND i_Interlocks[8];

// NETWORK 2
bCmdFwd := SEL(i_ServiceMode, i_AutoCmdFwd, i_ManCmdFwd);

// NETWORK 3
bCmdBwd := SEL(i_ServiceMode, i_AutoCmdBwd, i_ManCmdBwd);

// NETWORK 4
q_SpeedSP := SEL(i_ServiceMode, i_AutoSpeedSP, i_ManSpeedSP);

// NETWORK 5
tonBcwOff(IN := NOT bCmdBwd, PT := T#1s); // TON
tofCMDFwd(IN := q_InterlocksOK AND bCmdFwd AND tonBcwOff.Q, PT := T#100ms); // TOF
q_bCmdFwd := tofCMDFwd.Q;

// NETWORK 6
tonFwdOff(IN := NOT bCmdFwd, PT := T#1s); // TON
tofCMDBwd(IN := q_InterlocksOK AND bCmdBwd AND tonFwdOff.Q, PT := T#100ms); // TOF
q_bCmdBwd := tofCMDBwd.Q;

// NETWORK 7
_w1 := NOT i_ServiceMode OR i_ManStop;
i_ManCmdFwd R= _w1;
i_ManCmdBwd R= _w1;

// NETWORK 8
i_ManStop R= TRUE;

// NETWORK 9 (disabled)
// label: Feedback monitoring

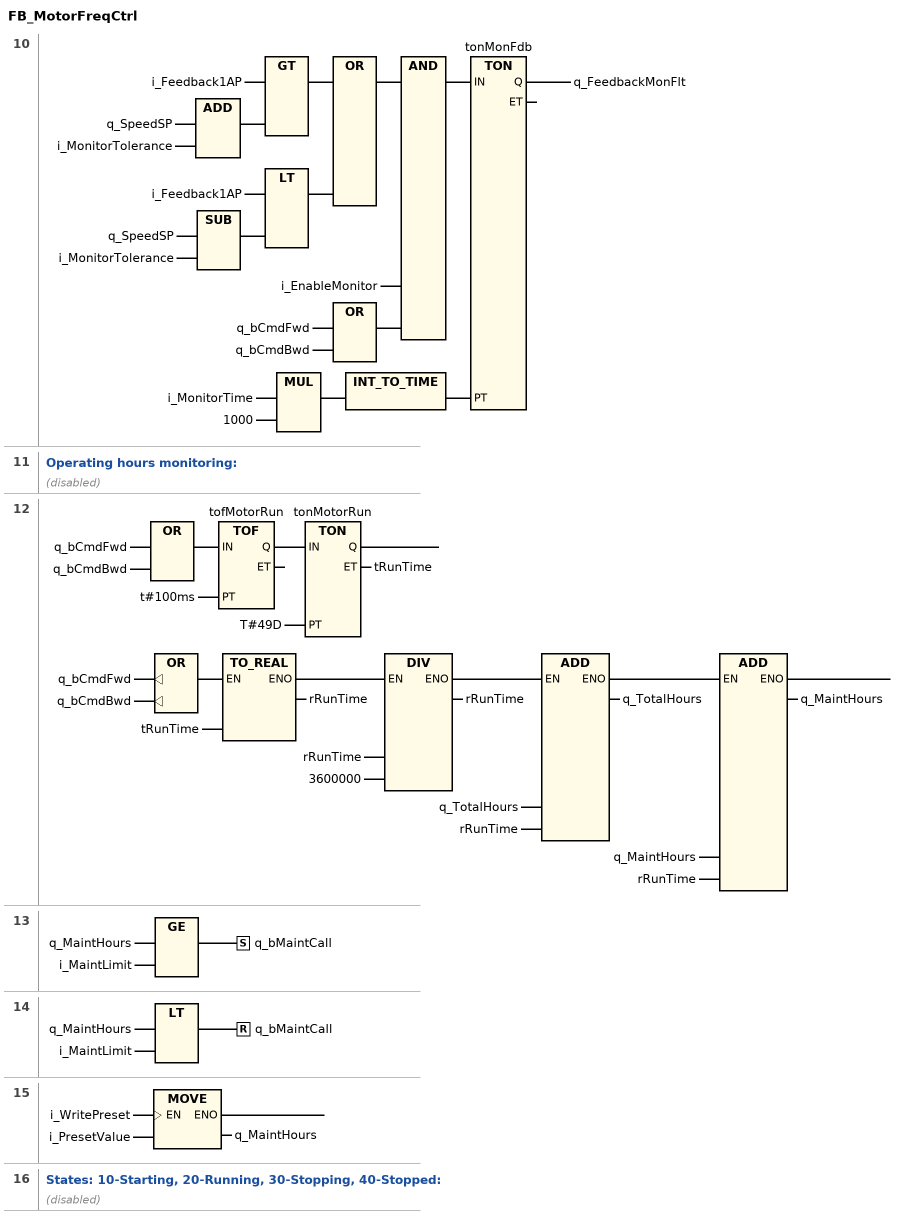
// NETWORK 10
tonMonFdb(IN := (i_Feedback1AP > q_SpeedSP + i_MonitorTolerance OR i_Feedback1AP < q_SpeedSP - i_MonitorTolerance) AND i_EnableMonitor AND (q_bCmdFwd OR q_bCmdBwd), PT := INT_TO_TIME(i_MonitorTime * 1000)); // TON
q_FeedbackMonFlt := tonMonFdb.Q;

// NETWORK 11 (disabled)
// label: Operating hours monitoring

// NETWORK 12
tofMotorRun(IN := q_bCmdFwd OR q_bCmdBwd, PT := t#100ms); // TOF
tonMotorRun(IN := tofMotorRun.Q, PT := T#49D, ET => tRunTime); // TON
_ft1(CLK := q_bCmdFwd);
_ft2(CLK := q_bCmdBwd);
_w2 := _ft1.Q OR _ft2.Q;
IF _w2 THEN rRunTime := TO_REAL(tRunTime); END_IF
IF _w2 THEN rRunTime := rRunTime / 3600000; END_IF
IF _w2 THEN q_TotalHours := q_TotalHours + rRunTime; END_IF
IF _w2 THEN q_MaintHours := q_MaintHours + rRunTime; END_IF

// NETWORK 13
q_bMaintCall S= q_MaintHours >= i_MaintLimit;

// NETWORK 14
q_bMaintCall R= q_MaintHours < i_MaintLimit;

// NETWORK 15
_rt1(CLK := i_WritePreset);
IF _rt1.Q THEN q_MaintHours := i_PresetValue; END_IF

// NETWORK 16 (disabled)
// label: States: 10-Starting, 20-Running, 30-Stopping, 40-Stopped

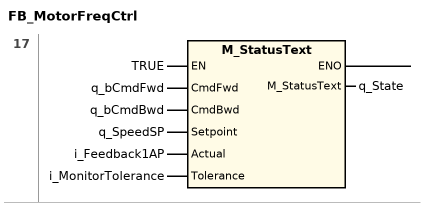
// NETWORK 17
q_State := M_StatusText(CmdFwd := q_bCmdFwd, CmdBwd := q_bCmdBwd, Setpoint := q_SpeedSP, Actual := i_Feedback1AP, Tolerance := i_MonitorTolerance);

METHOD M_StatusText : INT
VAR_INPUT
	CmdFwd		:BOOL;
	CmdBwd		:BOOL;
	Setpoint	:REAL;
	Actual		:REAL;
	Tolerance	:INT;
END_VAR
IF (CmdFwd OR CmdBwd) AND (Actual <= Setpoint-Tolerance+1) THEN
	M_StatusText := 10;	//Starting
ELSIF (CmdFwd OR CmdBwd) AND (Actual >= Setpoint-Tolerance+1) AND (Actual <= Setpoint+Tolerance+1) THEN
	M_StatusText := 20;	//Running
ELSIF (NOT CmdFwd AND NOT CmdBwd) AND (Actual >= 0+Tolerance+1) THEN
	M_StatusText := 30;	//Stopping
ELSIF (NOT CmdFwd AND NOT CmdBwd) AND (Actual <= 0+Tolerance+1)
		OR (NOT CmdFwd AND NOT CmdBwd) AND Setpoint >= Actual THEN
	M_StatusText := 40;	//Stopped
END_IF
END_METHOD

END_FUNCTION_BLOCK

// ---- FBs/Devices/FB_AnalogOutput_v01.TcPOU
// Created by Dimitar Stojanov 06.2023 

//Functionality: Use this block to scale Analog Outputs

FUNCTION_BLOCK FB_AnalogOutput_v01
VAR_INPUT
	i_rValue 							:REAL;
	i_rData_Low 						:REAL;
	i_rData_High 						:REAL;
	i_rScaled_Low						:INT	:=0;
	i_rScaled_High						:INT	:=32676;
	
END_VAR
VAR_OUTPUT
	q_iScaled							:INT;
END_VAR
VAR
	K								    :REAL;
END_VAR

K := ((i_rScaled_High - i_rScaled_Low) / (i_rData_High - i_rData_Low));
q_iScaled:=REAL_TO_INT(K * i_rValue);

END_FUNCTION_BLOCK

// ---- FBs/Devices/FB_MotorCoilsCtrl.TcPOU
FUNCTION_BLOCK FB_MotorCoilsCtrl
VAR_INPUT
	i_Interlocks		:ARRAY[1..8] OF BOOL;
	i_AutoCmdSlow		:BOOL;
	i_AutoCmdFast		:BOOL;
	i_ManCmdSlow		:BOOL;
	i_ManCmdFast		:BOOL;
	i_ManStop			:BOOL;
	i_SlowSpeed			:REAL;
	i_FastSpeed			:REAL;
	i_Feedback1AP		:REAL;
	i_Feedback2AP		:REAL;
	i_EnableMonitor		:BOOL;
	i_MonitorTime		:INT;
	i_MonitorTolerance	:INT;
	i_ServiceMode		:BOOL;
	i_MaintLimit		:REAL;
	i_PresetValue		:REAL;
	i_WritePreset		:BOOL;
END_VAR
VAR_OUTPUT
	q_InterlocksOK		:BOOL;
	q_bCmdSlow			:BOOL;
	q_bCmdFast			:BOOL;
	q_FeedbackMonFlt	:BOOL;
	q_TotalHours		:REAL;
	q_MaintHours		:REAL;
	q_bMaintCall		:BOOL;	
	q_State				:INT;
END_VAR
VAR
	bInTolerance		:BOOL;
	tRunTime			:TIME;
	rRunTime			:REAL;
	tonMonFdb			:TON;
	tonMotorRun			:TON;
	tofMotorRun			:TOF;
END_VAR
VAR // added by the converter: edge detectors and wires of the graphical bodies
    _w1, _w2 : BOOL;
    _ft1, _ft2 : F_TRIG;
    _rt1 : R_TRIG;
END_VAR

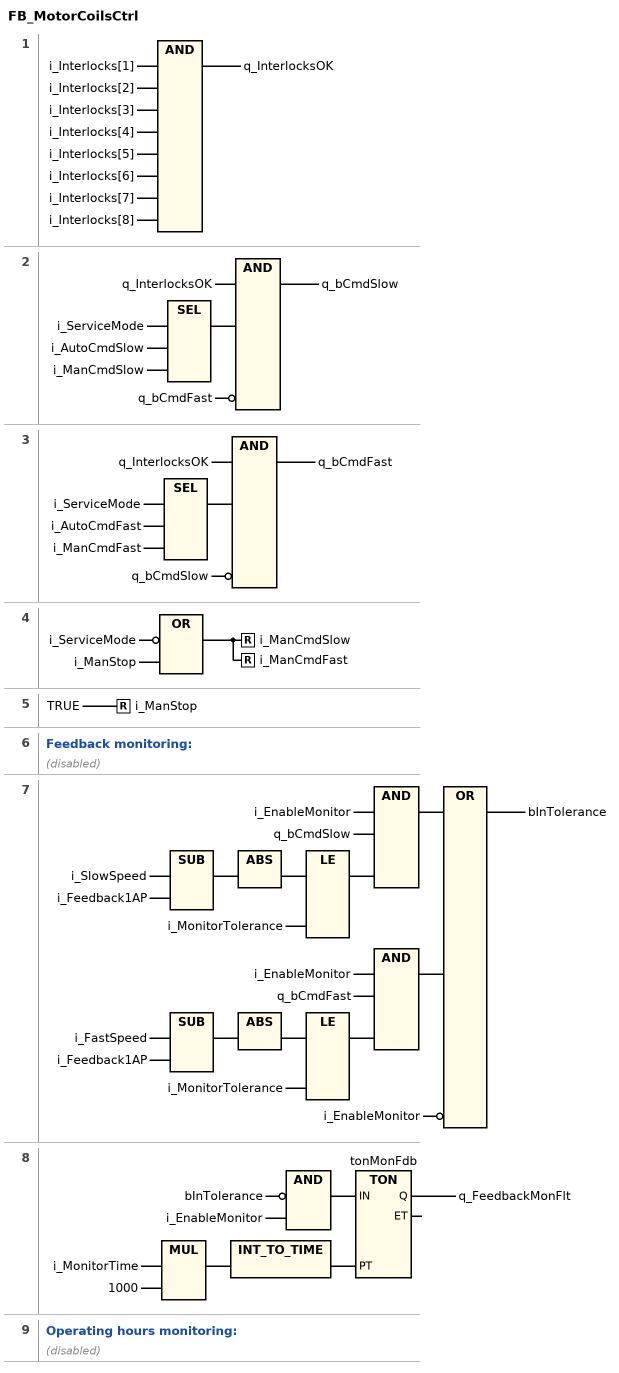
// NETWORK 1
q_InterlocksOK := i_Interlocks[1] AND i_Interlocks[2] AND i_Interlocks[3] AND i_Interlocks[4] AND i_Interlocks[5] AND i_Interlocks[6] AND i_Interlocks[7] AND i_Interlocks[8];

// NETWORK 2
q_bCmdSlow := q_InterlocksOK AND SEL(i_ServiceMode, i_AutoCmdSlow, i_ManCmdSlow) AND NOT q_bCmdFast;

// NETWORK 3
q_bCmdFast := q_InterlocksOK AND SEL(i_ServiceMode, i_AutoCmdFast, i_ManCmdFast) AND NOT q_bCmdSlow;

// NETWORK 4
_w1 := NOT i_ServiceMode OR i_ManStop;
i_ManCmdSlow R= _w1;
i_ManCmdFast R= _w1;

// NETWORK 5
i_ManStop R= TRUE;

// NETWORK 6 (disabled)
// label: Feedback monitoring

// NETWORK 7
bInTolerance := i_EnableMonitor AND q_bCmdSlow AND ABS(i_SlowSpeed - i_Feedback1AP) <= i_MonitorTolerance OR i_EnableMonitor AND q_bCmdFast AND ABS(i_FastSpeed - i_Feedback1AP) <= i_MonitorTolerance OR NOT i_EnableMonitor;

// NETWORK 8
tonMonFdb(IN := NOT bInTolerance AND i_EnableMonitor, PT := INT_TO_TIME(i_MonitorTime * 1000)); // TON
q_FeedbackMonFlt := tonMonFdb.Q;

// NETWORK 9 (disabled)
// label: Operating hours monitoring

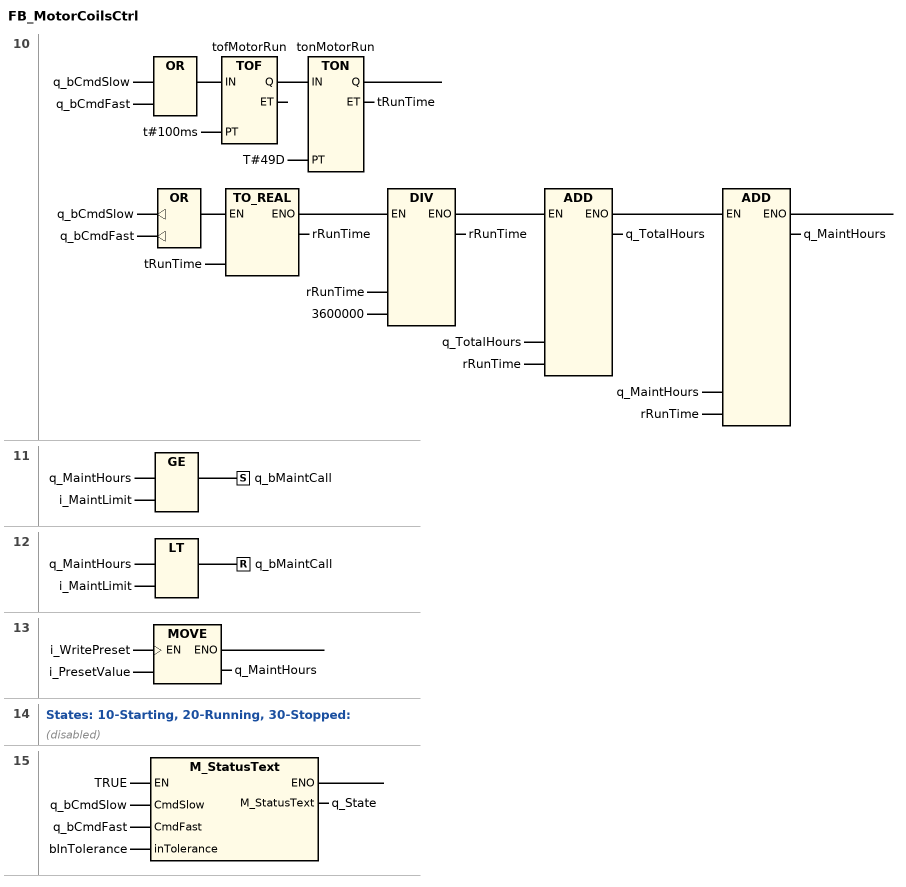
// NETWORK 10
tofMotorRun(IN := q_bCmdSlow OR q_bCmdFast, PT := t#100ms); // TOF
tonMotorRun(IN := tofMotorRun.Q, PT := T#49D, ET => tRunTime); // TON
_ft1(CLK := q_bCmdSlow);
_ft2(CLK := q_bCmdFast);
_w2 := _ft1.Q OR _ft2.Q;
IF _w2 THEN rRunTime := TO_REAL(tRunTime); END_IF
IF _w2 THEN rRunTime := rRunTime / 3600000; END_IF
IF _w2 THEN q_TotalHours := q_TotalHours + rRunTime; END_IF
IF _w2 THEN q_MaintHours := q_MaintHours + rRunTime; END_IF

// NETWORK 11
q_bMaintCall S= q_MaintHours >= i_MaintLimit;

// NETWORK 12
q_bMaintCall R= q_MaintHours < i_MaintLimit;

// NETWORK 13
_rt1(CLK := i_WritePreset);
IF _rt1.Q THEN q_MaintHours := i_PresetValue; END_IF

// NETWORK 14 (disabled)
// label: States: 10-Starting, 20-Running, 30-Stopped

// NETWORK 15
q_State := M_StatusText(CmdSlow := q_bCmdSlow, CmdFast := q_bCmdFast, inTolerance := bInTolerance);

METHOD M_StatusText : INT
VAR_INPUT
	CmdSlow		:BOOL;
	CmdFast		:BOOL;
	inTolerance	:BOOL;
END_VAR
IF (CmdSlow OR CmdFast) AND NOT inTolerance THEN
	M_StatusText := 10;	//Starting
ELSIF (CmdSlow OR CmdFast) AND inTolerance THEN
	M_StatusText := 20;	//Running
ELSIF (NOT CmdSlow AND NOT CmdFast) THEN
	M_StatusText := 30;	//Stopped
END_IF
END_METHOD

END_FUNCTION_BLOCK

// ---- FBs/Devices/FB_CoilCtrl.TcPOU
FUNCTION_BLOCK FB_CoilCtrl
VAR_INPUT
	i_Interlocks		:ARRAY[1..8] OF BOOL;
	i_ProcesslocksOK	:BOOL;
	i_AutoCmd			:BOOL;
	i_ManCmd			:BOOL;
	i_ServiceMode		:BOOL;
	i_MaintLimit		:UDINT;
	i_PresetValue		:UDINT;
	i_WritePreset		:BOOL;
END_VAR
VAR_OUTPUT
	q_InterlocksOK		:BOOL;
	q_Enabled			:BOOL;
	q_Cmd				:BOOL;
	q_TotalCycles		:UDINT;
	q_MaintCycles		:UDINT;
	q_MaintenanceCall	:BOOL;
END_VAR
VAR
	tofDelayOut			:TOF;
	bCmd				:BOOL;
END_VAR
VAR // added by the converter: edge detectors and wires of the graphical bodies
    _rt1, _rt2 : R_TRIG;
    _w1 : BOOL;
END_VAR

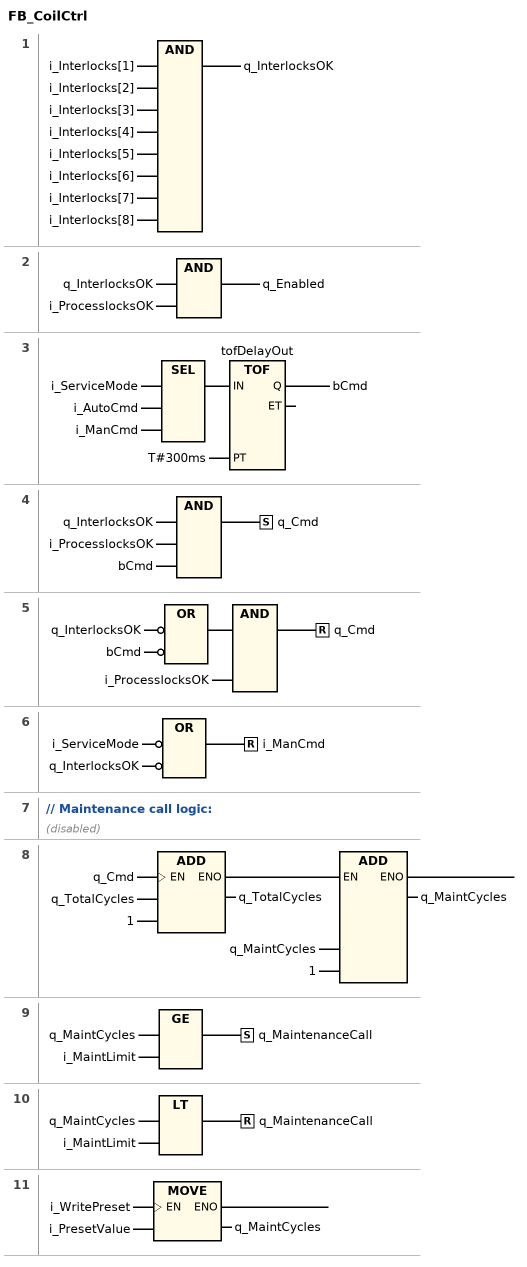
// NETWORK 1
q_InterlocksOK := i_Interlocks[1] AND i_Interlocks[2] AND i_Interlocks[3] AND i_Interlocks[4] AND i_Interlocks[5] AND i_Interlocks[6] AND i_Interlocks[7] AND i_Interlocks[8];

// NETWORK 2
q_Enabled := q_InterlocksOK AND i_ProcesslocksOK;

// NETWORK 3
tofDelayOut(IN := SEL(i_ServiceMode, i_AutoCmd, i_ManCmd), PT := T#300ms); // TOF
bCmd := tofDelayOut.Q;

// NETWORK 4
q_Cmd S= q_InterlocksOK AND i_ProcesslocksOK AND bCmd;

// NETWORK 5
q_Cmd R= (NOT q_InterlocksOK OR NOT bCmd) AND i_ProcesslocksOK;

// NETWORK 6
i_ManCmd R= NOT i_ServiceMode OR NOT q_InterlocksOK;

// NETWORK 7 (disabled)
// label: // Maintenance call logic

// NETWORK 8
_rt1(CLK := q_Cmd);
_w1 := _rt1.Q;
IF _w1 THEN q_TotalCycles := q_TotalCycles + 1; END_IF
IF _w1 THEN q_MaintCycles := q_MaintCycles + 1; END_IF

// NETWORK 9
q_MaintenanceCall S= q_MaintCycles >= i_MaintLimit;

// NETWORK 10
q_MaintenanceCall R= q_MaintCycles < i_MaintLimit;

// NETWORK 11
_rt2(CLK := i_WritePreset);
IF _rt2.Q THEN q_MaintCycles := i_PresetValue; END_IF

END_FUNCTION_BLOCK

// ---- FBs/Devices/FB_PID.TcPOU
FUNCTION_BLOCK FB_PID
VAR_INPUT
	i_bEnablePID		:BOOL	:=FALSE;
	i_rSetpoint			:REAL;				//required input from PLC logic
	i_rActual			:REAL;				//required input from PLC logic
	i_rKp				:REAL;
	i_rKi				:REAL;
	i_rKd				:REAL;
	i_rTdamp			:REAL;
	i_rOutMin			:REAL	:=0;
	i_rOutMax			:REAL	:=100;
	i_rManualOutput		:REAL	:=0;
	i_bEnablePWM		:BOOL	:=FALSE;
	i_iFreqPWM			:INT	:=1000;		//required input from PLC logic
	i_bAutotuneStart	:BOOL	:=FALSE;
	i_rAutotuneSetpoint	:REAL	:=0;
	i_bEnableAlarms		:BOOL;
	i_iHighAlarm		:INT;
	i_iHighWarning		:INT;
	i_iLowWarning		:INT;
	i_iLowAlarm			:INT;
	i_iWarningDelay		:INT;
	i_iAlarmDelay		:INT;
END_VAR
VAR_OUTPUT
	q_rOutputPID		:REAL;				//output for proportional control
	q_bOutputPWM		:BOOL;				//output for on/off control
	q_Difference		:REAL;
	q_AutotuneActive	:BOOL;
	q_AutotuneDone		:BOOL;
	i_sAutotuneTime		:STRING	:='00:00:00';
	q_rAutotuneKp		:REAL	:=0;
	q_rAutotuneKi		:REAL	:=0;
	q_rAutotuneKd		:REAL	:=0;
	q_bError			:BOOL;
	q_bErrorID			:INT	:=0;;
	q_bAlarmHigh		:BOOL;				
	q_bWarningHigh		:BOOL;
	q_bWarningLow		:BOOL;
	q_bAlarmLow			:BOOL;
END_VAR
VAR
	PID_AutoTuner		:FB_PID_AutoTuner;
	PWM_Autotune		:FB_PID_PWM;
	PID_Gain2Time		:FB_PID_Gain2Time;
	ST_PID_Params		:ST_CTRL_PID_PARAMS;
	PID_Control			:FB_CTRL_PID;
	PWM_Control			:FB_PID_PWM;
	M_Active_0			:FB_CTRL_PID;
	
	tonAlarmHigh		:TON;
	tonWarningHigh		:TON;
	tonWarningLow		:TON;
	tonAlarmLow			:TON;
	tonAutotuneTime		:TON;
	
END_VAR
VAR // added by the converter: edge detectors and wires of the graphical bodies
    _w1, _w2, _w3, _w4, _w5 : BOOL;
END_VAR

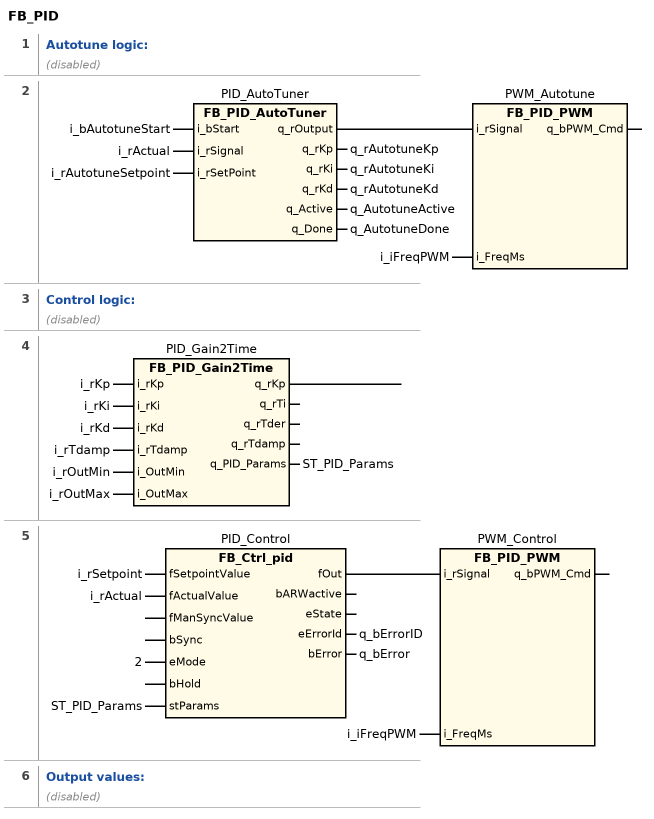
// NETWORK 1 (disabled)
// label: Autotune logic

// NETWORK 2
PID_AutoTuner(
    i_bStart := i_bAutotuneStart,
    i_rSignal := i_rActual,
    i_rSetPoint := i_rAutotuneSetpoint,
    q_rKp => q_rAutotuneKp,
    q_rKi => q_rAutotuneKi,
    q_rKd => q_rAutotuneKd,
    q_Active => q_AutotuneActive,
    q_Done => q_AutotuneDone); // FB_PID_AutoTuner
PWM_Autotune(i_rSignal := PID_AutoTuner.q_rOutput, i_FreqMs := i_iFreqPWM); // FB_PID_PWM

// NETWORK 3 (disabled)
// label: Control logic

// NETWORK 4
PID_Gain2Time(
    i_rKp := i_rKp,
    i_rKi := i_rKi,
    i_rKd := i_rKd,
    i_rTdamp := i_rTdamp,
    i_OutMin := i_rOutMin,
    i_OutMax := i_rOutMax,
    q_PID_Params => ST_PID_Params); // FB_PID_Gain2Time

// NETWORK 5
PID_Control(
    fSetpointValue := i_rSetpoint,
    fActualValue := i_rActual,
    eMode := 2,
    stParams := ST_PID_Params,
    eErrorId => q_bErrorID,
    bError => q_bError); // FB_Ctrl_pid
PWM_Control(i_rSignal := PID_Control.fOut, i_FreqMs := i_iFreqPWM); // FB_PID_PWM

// NETWORK 6 (disabled)
// label: Output values

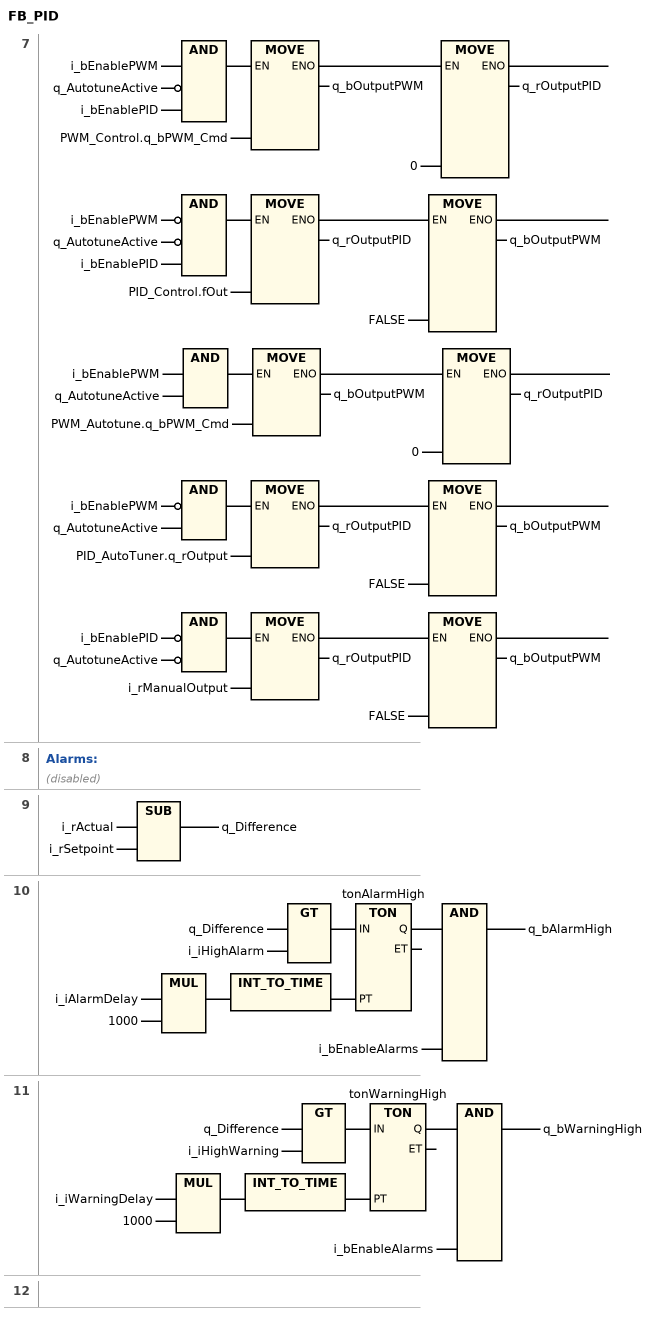
// NETWORK 7
_w1 := i_bEnablePWM AND NOT q_AutotuneActive AND i_bEnablePID;
IF _w1 THEN q_bOutputPWM := PWM_Control.q_bPWM_Cmd; END_IF
IF _w1 THEN q_rOutputPID := 0; END_IF
_w2 := NOT i_bEnablePWM AND NOT q_AutotuneActive AND i_bEnablePID;
IF _w2 THEN q_rOutputPID := PID_Control.fOut; END_IF
IF _w2 THEN q_bOutputPWM := FALSE; END_IF
_w3 := i_bEnablePWM AND q_AutotuneActive;
IF _w3 THEN q_bOutputPWM := PWM_Autotune.q_bPWM_Cmd; END_IF
IF _w3 THEN q_rOutputPID := 0; END_IF
_w4 := NOT i_bEnablePWM AND q_AutotuneActive;
IF _w4 THEN q_rOutputPID := PID_AutoTuner.q_rOutput; END_IF
IF _w4 THEN q_bOutputPWM := FALSE; END_IF
_w5 := NOT i_bEnablePID AND NOT q_AutotuneActive;
IF _w5 THEN q_rOutputPID := i_rManualOutput; END_IF
IF _w5 THEN q_bOutputPWM := FALSE; END_IF

// NETWORK 8 (disabled)
// label: Alarms

// NETWORK 9
q_Difference := i_rActual - i_rSetpoint;

// NETWORK 10
tonAlarmHigh(IN := q_Difference > i_iHighAlarm, PT := INT_TO_TIME(i_iAlarmDelay * 1000)); // TON
q_bAlarmHigh := tonAlarmHigh.Q AND i_bEnableAlarms;

// NETWORK 11
tonWarningHigh(IN := q_Difference > i_iHighWarning, PT := INT_TO_TIME(i_iWarningDelay * 1000)); // TON
q_bWarningHigh := tonWarningHigh.Q AND i_bEnableAlarms;

// NETWORK 12

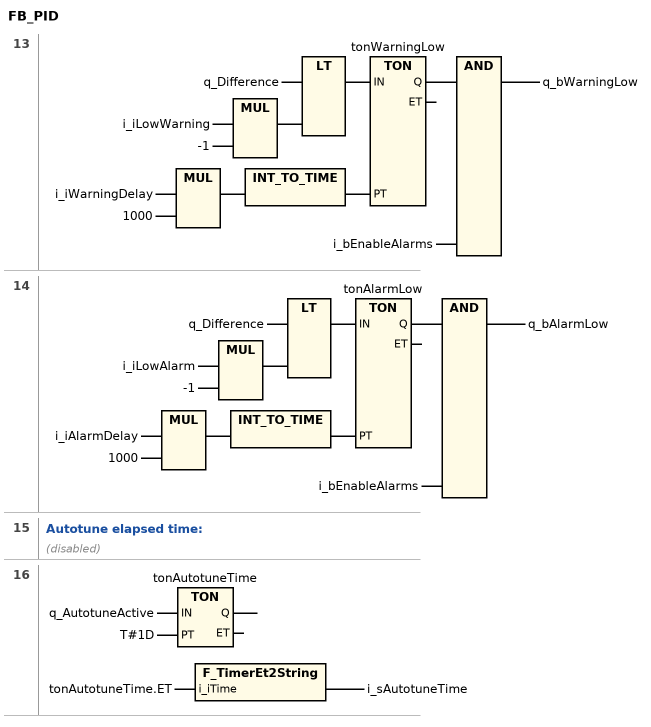
// NETWORK 13
tonWarningLow(IN := q_Difference < i_iLowWarning * -1, PT := INT_TO_TIME(i_iWarningDelay * 1000)); // TON
q_bWarningLow := tonWarningLow.Q AND i_bEnableAlarms;

// NETWORK 14
tonAlarmLow(IN := q_Difference < i_iLowAlarm * -1, PT := INT_TO_TIME(i_iAlarmDelay * 1000)); // TON
q_bAlarmLow := tonAlarmLow.Q AND i_bEnableAlarms;

// NETWORK 15 (disabled)
// label: Autotune elapsed time

// NETWORK 16
tonAutotuneTime(IN := q_AutotuneActive, PT := T#1D); // TON
i_sAutotuneTime := F_TimerEt2String(i_iTime := tonAutotuneTime.ET);

END_FUNCTION_BLOCK

// ---- FBs/Devices/FB_PID_AutoTuner.TcPOU
FUNCTION_BLOCK FB_PID_AutoTuner
VAR_INPUT
	i_bStart					:BOOL;
	i_rSignal					:REAL;
	i_rSetPoint					:REAL;
END_VAR

VAR_OUTPUT			
	q_rOutput					:REAL;
	q_rKp						:REAL;
	q_rKi						:REAL;
	q_rKd						:REAL;
	q_Active					:BOOL;
	q_Done						:BOOL;
END_VAR

VAR
	rPeakMax					:REAL;	
	rPrevMax					:REAL:=1;
	rPeakMin					:REAL;
	rPrevMin					:REAL:=0;
	tPrevPeriod					:TIME;
	tNewPeriod					:TIME;
	tonPeriodTimer				:TON;
	iStep						:INT:=0;
	rtrigStart					:R_TRIG;
END_VAR

rtrigStart(CLK:=i_bStart);

IF NOT i_bStart THEN
	iStep := 0;
END_IF

//Output - autotune active
IF iStep <> 0 THEN	
	q_Active := TRUE; 
ELSE 
	q_Active := FALSE; 
END_IF
	
//Output - autotune done
IF iStep=700 THEN 
	q_Done:=TRUE; 
ELSIF iStep=50 THEN 
	q_Done:=FALSE; 
END_IF

CASE iStep OF 
	//start pod setpoint
	0:
		rPeakMax:=i_rSetPoint;
		rPeakMin:=i_rSetPoint;
		rPrevMax:=i_rSetPoint;
		rPrevMin:=0;
		tPrevPeriod:=T#1ms;
		IF rtrigStart.Q THEN
			iStep := 50;
		END_IF
		
	50:
		q_rKp := 1;
		q_rKi := 1;
		q_rKd := 1;
		iStep := 100;
		
	100: 
		IF i_rSignal > i_rSetPoint THEN
			iStep := 200;
		END_IF
		
	//nad setpoint
	200: 
		IF i_rSignal >= rPeakMax THEN
			rPeakMax := i_rSignal;
		END_IF
		
		IF i_rSignal < i_rSetPoint THEN
				iStep := 300;
		END_IF
	
	//pod setpoint
	300:
		IF i_rSignal <= rPeakMin THEN
			rPeakMin := i_rSignal;
		END_IF
		IF i_rSignal > i_rSetPoint THEN
			iStep := 400;
		END_IF
		
	//proverka za da ne delime so 0
	400: 
		IF tPrevPeriod <> T#0MS AND (rPrevMax-rPrevMin) <> 0 THEN
			iStep := 500;
		ELSE
			rPeakMax := i_rSetpoint;
			rPeakMin := i_rSetpoint;
			iStep := 200;
		END_IF
		
	//compare
	500:
		IF (ABS(((rPeakMax-rPeakMin) - (rPrevMax-rPrevMin))/(rPrevMax-rPrevMin)) <= (0.1)) AND (ABS(TIME_TO_REAL(tNewPeriod) - TIME_TO_REAL(tPrevPeriod))/TIME_TO_REAL(tPrevPeriod) <= (0.1)) THEN 
			iStep := 600;
		ELSE
			rPrevMax := rPeakMax;
			rPrevMin := rPeakMin;
			rPeakMax := i_rSetpoint;
			rPeakMin := i_rSetpoint;
			
			tPrevPeriod := tNewPeriod;
			iStep := 200;
		END_IF
	
	//presmetki PID
	600:
		q_rKp := 0.35*4*100/(PI*(rPeakMax-rPeakMin));
		q_rKi := 1.85*4*100/(PI*(rPeakMax-rPeakMin))/(TIME_TO_REAL(tNewPeriod)/1000); 
		q_rKd := 0.05*4*100/(PI*(rPeakMax-rPeakMin))*(TIME_TO_REAL(tNewPeriod)/1000); 
		iStep := 700;
		
	700:
		iStep := 0;
	
END_CASE

IF (iStep=100 OR iStep=300) THEN
	q_rOutput := 100;
ELSE
	q_rOutput := 0;
END_IF

tonPeriodTimer(IN := (iStep>=100 AND iStep<=300), PT := T#15H);
IF tonPeriodTimer.IN THEN
	tNewPeriod := tonPeriodTimer.ET;
END_IF

END_FUNCTION_BLOCK

// ---- FBs/Devices/FB_PID_PWM.TcPOU
FUNCTION_BLOCK FB_PID_PWM
VAR_INPUT
	i_rSignal					:REAL;
	i_FreqMs					:REAL;
END_VAR
VAR_OUTPUT
	q_bPWM_Cmd					:BOOL;
END_VAR
VAR
	tonSignalOFF				:TON;
	tofSignalON					:TOF;
	Multiplier					:REAL;
END_VAR

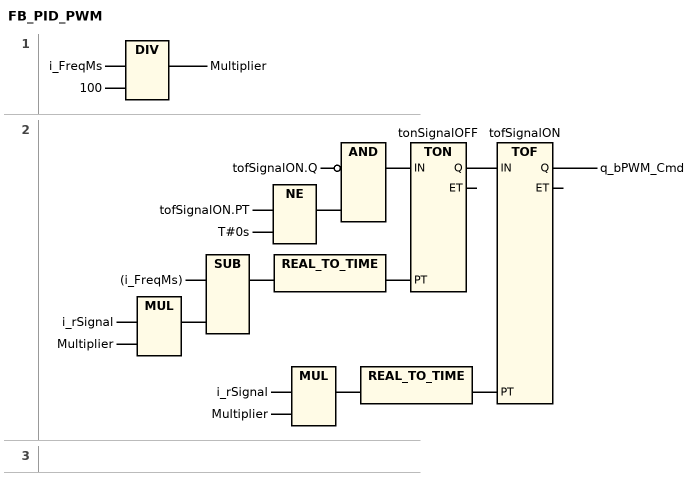
// NETWORK 1
Multiplier := i_FreqMs / 100;

// NETWORK 2
tonSignalOFF(IN := NOT tofSignalON.Q AND tofSignalON.PT <> T#0s, PT := REAL_TO_TIME(((i_FreqMs)) - i_rSignal * Multiplier)); // TON
tofSignalON(IN := tonSignalOFF.Q, PT := REAL_TO_TIME(i_rSignal * Multiplier)); // TOF
q_bPWM_Cmd := tofSignalON.Q;

// NETWORK 3

END_FUNCTION_BLOCK

// ---- FBs/Devices/FB_PID_Gain2Time.TcPOU
FUNCTION_BLOCK FB_PID_Gain2Time
VAR_INPUT
	i_rKp					:REAL;
	i_rKi					:REAL;
	i_rKd					:REAL;
	i_rTdamp				:REAL := 10;
	i_OutMin				:REAL := 0;
	i_OutMax				:REAL := 100;
END_VAR

VAR_OUTPUT
	q_rKp					:REAL;
	q_rTi					:REAL;
	q_rTder					:REAL;
	q_rTdamp				:REAL;
	
	q_PID_Params			:st_CTRL_pid_params;
END_VAR

//Limitation and validation rules
i_rKi := LIMIT(0.000000000001, i_rKi, 1000000);
i_rKp := LIMIT(0.000000000001, i_rKp, 1000000);
i_OutMin := LIMIT(0, i_OutMin, 100);
i_OutMax := LIMIT(0, i_OutMax, 100);
IF i_OutMin >= i_OutMax THEN
	i_OutMin := 0;
END_IF


q_rKp := i_rKp;
q_rTi := (i_rKp*0.01/i_rKi);
q_rTder := i_rKd/i_rKp;
q_rTdamp := i_rTdamp;

q_PID_Params.tCtrlCycleTime := T#10MS;
q_PID_Params.tTaskCycleTime := T#10MS;
q_PID_Params.fKp := q_rKp; //gain
q_PID_Params.tTn := REAL_TO_TIME(q_rTi*1000);
q_PID_Params.tTv := REAL_TO_TIME(q_rTder*1000); //derivative
q_PID_Params.tTd := REAL_TO_TIME(q_rTder*1000); //dampening
q_PID_Params.fOutMinLimit := i_OutMin;
q_PID_Params.fOutMaxLimit := i_OutMax;

END_FUNCTION_BLOCK

// ---- Functions/F_TimerEt2String.TcPOU
FUNCTION F_TimerEt2String : STRING
VAR_INPUT
	i_iTime				:TIME;
END_VAR
VAR
	iTimeInSec			:UDINT;
	iHours				:UDINT;
	iMinutes			:UDINT;
	iSeconds			:UDINT;
	sQuery				:STRING;
END_VAR

iTimeInSec:=TO_UDINT(i_iTIme)/1000;

iHours:=iTimeInSec/3600;
iMinutes:=(iTimeInSec/60)-(iHours*60);
iSeconds:=iTimeInSec - (iMinutes*60) - (iHours*3600);

IF iHours = 0 THEN
	sQuery:='00:';
ELSIF iHours > 0 AND iHours < 10 THEN
	sQuery:=CONCAT('0',TO_STRING(iHours));
	sQuery:=CONCAT(sQuery,':');
ELSE
	sQuery:=TO_STRING(iHours);
	sQuery:=CONCAT(sQuery,':');
END_IF

IF iMinutes = 0 THEN
	sQuery:=CONCAT(sQuery,'00:');
ELSIF iMinutes > 0 AND iMinutes < 10 THEN
	sQuery:=CONCAT(sQuery,'0');
	sQuery:=CONCAT(sQuery,TO_STRING(iMinutes));
	sQuery:=CONCAT(sQuery,':');
ELSE
	sQuery:=CONCAT(sQuery,TO_STRING(iMinutes));
	sQuery:=CONCAT(sQuery,':');
END_IF

IF iSeconds = 0 THEN
	sQuery:=CONCAT(sQuery,'00');
ELSIF iSeconds > 0 AND iSeconds < 10 THEN
	sQuery:=CONCAT(sQuery,'0');
	sQuery:=CONCAT(sQuery,TO_STRING(iSeconds));
ELSE
	sQuery:=CONCAT(sQuery,TO_STRING(iSeconds));
END_IF


F_TimerEt2String:=sQuery;

END_FUNCTION

// ---- FBs/Devices/FB_AnalogOutput_v02.TcPOU
FUNCTION_BLOCK FB_AnalogOutput_v02
VAR_INPUT
	i_rValue 							:REAL;
	i_rData_Low 						:REAL	:=0;
	i_rData_High 						:REAL	:=32676;
	i_rScaled_Low						:INT	:=0;
	i_rScaled_High						:INT	:=32676;
	i_rOffset 							:REAL;
	i_bSimToggle						:BOOL	:= FALSE;
	i_rSimValue							:REAL	:= 0;
	i_bServiceMode						:BOOL;				//Required signal from logic
END_VAR
VAR_OUTPUT
	q_rValue							:REAL;
	q_iScaled							:INT;
	q_bSimActive						:BOOL;
END_VAR
VAR
	K								    :REAL;
END_VAR

//Validation rules (protect divide by zero)
IF i_rData_High - i_rData_Low = 0 THEN 	i_rData_High := i_rData_Low + 1; END_IF

//Simulation
q_bSimActive := i_bSimToggle AND i_bServiceMode;
IF NOT i_bServiceMode THEN i_bSimToggle := FALSE; END_IF

IF q_bSimActive THEN q_rValue := i_rSimValue + i_rOffset; ELSE q_rValue := i_rValue + i_rOffset; END_IF

//Scaling
K := ((i_rScaled_High - i_rScaled_Low) / (i_rData_High - i_rData_Low));
q_iScaled:=REAL_TO_INT(K * q_rValue);

END_FUNCTION_BLOCK

// ---- FBs/Devices/FB_ValveCtrl52.TcPOU
FUNCTION_BLOCK FB_ValveCtrl52
VAR_INPUT
	i_Interlocks		:ARRAY[1..8] OF BOOL;
	i_ProcesslocksOK	:BOOL;
	i_AutoCmdHP			:BOOL;
	i_AutoCmdWP			:BOOL;
	i_ManCmdHP			:BOOL;
	i_ManCmdWP			:BOOL;
	i_ServiceMode		:BOOL;
	i_EnableHP			:BOOL;
	i_EnableWP			:BOOL;
	i_HP				:BOOL;
	i_WP				:BOOL;
	i_Timeout			:INT;
	i_MaintLimit		:UDINT;
	i_PresetValue		:UDINT;
	i_WritePreset		:BOOL;
END_VAR
VAR_OUTPUT
	q_InterlocksOK		:BOOL;
	q_Enabled			:BOOL;
	q_CmdHP				:BOOL;
	q_CmdWP				:BOOL;
	q_Traveling			:BOOL;
	q_AtHP				:BOOL;
	q_AtWP				:BOOL;
	q_TimeoutHP			:BOOL;
	q_TimeoutWP			:BOOL;
	q_SensorsFlt		:BOOL;
	q_TotalCycles		:UDINT;
	q_MaintCycles		:UDINT;
	q_MaintenanceCall	:BOOL;
	q_State				:INT;
END_VAR
VAR
	tonTimeoutHP		:TON;
	tonTimeoutWP		:TON;
	tonSensorsFlt		:TON;
	tofDelayOutHP		:TOF;
	tofDelayOutWP		:TOF;
	bCmdHP				:BOOL;
	bCmdWP				:BOOL;
END_VAR
VAR // added by the converter: edge detectors and wires of the graphical bodies
    _w1, _w2, _w3, _w4 : BOOL;
    _rt1, _rt2 : R_TRIG;
END_VAR

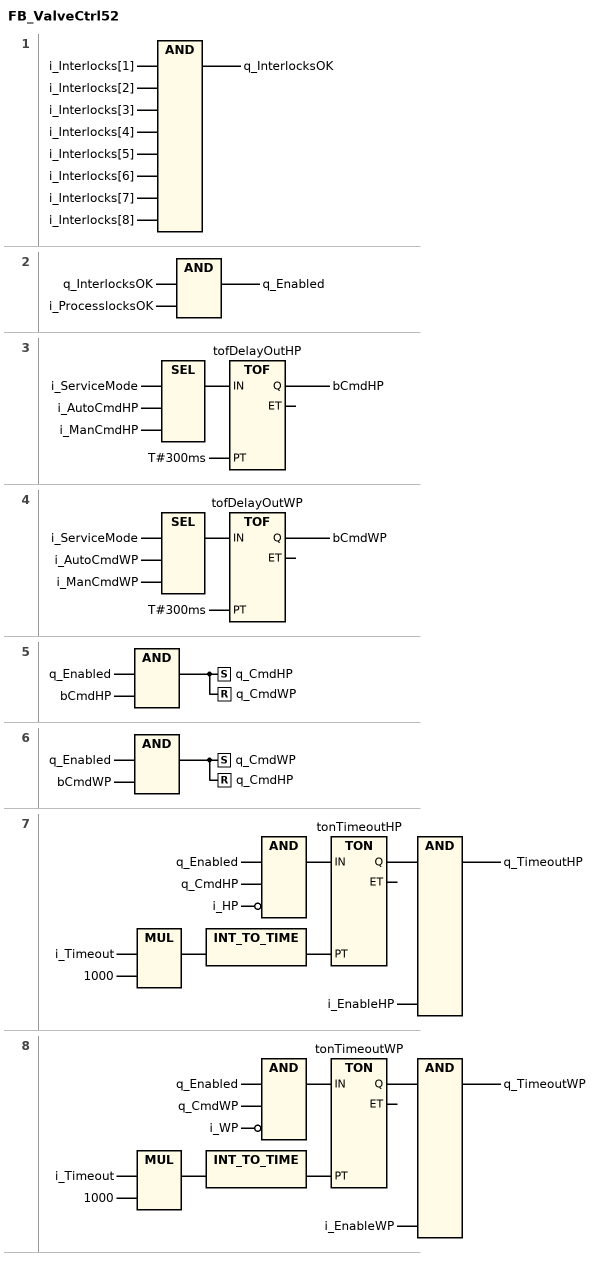
// NETWORK 1
q_InterlocksOK := i_Interlocks[1] AND i_Interlocks[2] AND i_Interlocks[3] AND i_Interlocks[4] AND i_Interlocks[5] AND i_Interlocks[6] AND i_Interlocks[7] AND i_Interlocks[8];

// NETWORK 2
q_Enabled := q_InterlocksOK AND i_ProcesslocksOK;

// NETWORK 3
tofDelayOutHP(IN := SEL(i_ServiceMode, i_AutoCmdHP, i_ManCmdHP), PT := T#300ms); // TOF
bCmdHP := tofDelayOutHP.Q;

// NETWORK 4
tofDelayOutWP(IN := SEL(i_ServiceMode, i_AutoCmdWP, i_ManCmdWP), PT := T#300ms); // TOF
bCmdWP := tofDelayOutWP.Q;

// NETWORK 5
_w1 := q_Enabled AND bCmdHP;
q_CmdHP S= _w1;
q_CmdWP R= _w1;

// NETWORK 6
_w2 := q_Enabled AND bCmdWP;
q_CmdWP S= _w2;
q_CmdHP R= _w2;

// NETWORK 7
tonTimeoutHP(IN := q_Enabled AND q_CmdHP AND NOT i_HP, PT := INT_TO_TIME(i_Timeout * 1000)); // TON
q_TimeoutHP := tonTimeoutHP.Q AND i_EnableHP;

// NETWORK 8
tonTimeoutWP(IN := q_Enabled AND q_CmdWP AND NOT i_WP, PT := INT_TO_TIME(i_Timeout * 1000)); // TON
q_TimeoutWP := tonTimeoutWP.Q AND i_EnableWP;

